LIN {X 0,Y 680.504,Z 396.458,A -85,B 0,C 180,E1 31291.838,E2 31291.838} C_VEL
LIN {X 0,Y 680.503,Z 396.457,A -85,B 0,C 180,E1 31288.855,E2 31288.855} C_VEL
LIN {X 0,Y 680.504,Z 396.449,A -85,B 0,C 180,E1 31285.651,E2 31285.651} C_VEL
LIN {X 0,Y 680.491,Z 396.449,A -85,B 0,C 180,E1 31282.744,E2 31282.744} C_VEL
LIN {X 0,Y 680.522,Z 396.462,A -85,B 0,C 180,E1 31279.612,E2 31279.612} C_VEL
LIN {X 0,Y 680.516,Z 396.57,A -85,B 0,C 180,E1 31279.434,E2 31279.434} C_VEL
LIN {X 0,Y 681.817,Z 400,A -85,B 0,C 180,E1 31279.04,E2 31279.04} C_VEL
LIN {X 0,Y 686.968,Z 410.535,A -85,B 0,C 180,E1 31277.744,E2 31277.744} C_VEL
LIN {X 0,Y 694.908,Z 427.67,A -85,B 0,C 180,E1 31275.744,E2 31275.744} C_VEL
LIN {X 0,Y 695.922,Z 430.045,A -85,B 0,C 180,E1 31275.624,E2 31275.624} C_VEL
LIN {X 0,Y 700.828,Z 449.853,A -85,B 0,C 180,E1 31274.934,E2 31274.934} C_VEL
LIN {X 0,Y 698.454,Z 660.17,A -85,B 0,C 180,E1 31272.2,E2 31272.2} C_VEL
LIN {X 0,Y 696.119,Z 885.552,A -85,B 0,C 180,E1 31269.363,E2 31269.363} C_VEL
LIN {X 0,Y 695.544,Z 917.031,A -85,B 0,C 180,E1 31268.911,E2 31268.911} C_VEL
LIN {X 0,Y 694.786,Z 942.091,A -85,B 0,C 180,E1 31268.4,E2 31268.4} C_VEL
LIN {X 0,Y 693.903,Z 967.65,A -85,B 0,C 180,E1 31267.73,E2 31267.73} C_VEL
LIN {X 0,Y 692.788,Z 994.389,A -85,B 0,C 180,E1 31266.849,E2 31266.849} C_VEL
LIN {X 0,Y 691.794,Z 1015.288,A -85,B 0,C 180,E1 31266.036,E2 31266.036} C_VEL
LIN {X 0,Y 690.754,Z 1035.672,A -85,B 0,C 180,E1 31265.129,E2 31265.129} C_VEL
LIN {X 0,Y 689.674,Z 1055.667,A -85,B 0,C 180,E1 31264.122,E2 31264.122} C_VEL
LIN {X 0,Y 688.501,Z 1076.875,A -85,B 0,C 180,E1 31262.921,E2 31262.921} C_VEL
LIN {X 0,Y 687.033,Z 1101.872,A -85,B 0,C 180,E1 31261.306,E2 31261.306} C_VEL
LIN {X 0,Y 685.952,Z 1121.014,A -85,B 0,C 180,E1 31259.905,E2 31259.905} C_VEL
LIN {X 0,Y 684.924,Z 1139.979,A -85,B 0,C 180,E1 31258.366,E2 31258.366} C_VEL
LIN {X 0,Y 683.775,Z 1160.558,A -85,B 0,C 180,E1 31256.49,E2 31256.49} C_VEL
LIN {X 0,Y 682.966,Z 1177.027,A -85,B 0,C 180,E1 31254.809,E2 31254.809} C_VEL
LIN {X 0,Y 682.152,Z 1194.232,A -85,B 0,C 180,E1 31252.86,E2 31252.86} C_VEL
LIN {X 0,Y 681.475,Z 1210.147,A -85,B 0,C 180,E1 31250.801,E2 31250.801} C_VEL
LIN {X 0,Y 681.039,Z 1222.568,A -85,B 0,C 180,E1 31249.001,E2 31249.001} C_VEL
LIN {X 0,Y 680.648,Z 1234.891,A -85,B 0,C 180,E1 31246.993,E2 31246.993} C_VEL
LIN {X 0,Y 680.343,Z 1246.823,A -85,B 0,C 180,E1 31244.733,E2 31244.733} C_VEL
LIN {X 0,Y 680.159,Z 1255.781,A -85,B 0,C 180,E1 31242.742,E2 31242.742} C_VEL
LIN {X 0,Y 680.022,Z 1262.732,A -85,B 0,C 180,E1 31240.937,E2 31240.937} C_VEL
LIN {X 0,Y 679.93,Z 1268.298,A -85,B 0,C 180,E1 31239.227,E2 31239.227} C_VEL
LIN {X 0,Y 679.925,Z 1273.362,A -85,B 0,C 180,E1 31237.354,E2 31237.354} C_VEL
LIN {X 0,Y 679.917,Z 1277.922,A -85,B 0,C 180,E1 31235.066,E2 31235.066} C_VEL
LIN {X 0,Y 679.912,Z 1280.606,A -85,B 0,C 180,E1 31232.87,E2 31232.87} C_VEL
LIN {X 0,Y 679.875,Z 1281.736,A -85,B 0,C 180,E1 31231.015,E2 31231.015} C_VEL
LIN {X 0,Y 679.863,Z 1281.828,A -85,B 0,C 180,E1 31229.33,E2 31229.33} C_VEL
LIN {X 0,Y 679.906,Z 1280.949,A -85,B 0,C 180,E1 31227.56,E2 31227.56} C_VEL
LIN {X 0,Y 679.915,Z 1278.924,A -85,B 0,C 180,E1 31225.618,E2 31225.618} C_VEL
LIN {X 0,Y 679.927,Z 1274.915,A -85,B 0,C 180,E1 31223.333,E2 31223.333} C_VEL
LIN {X 0,Y 679.942,Z 1269.344,A -85,B 0,C 180,E1 31221.122,E2 31221.122} C_VEL
LIN {X 0,Y 680.018,Z 1263.372,A -85,B 0,C 180,E1 31219.242,E2 31219.242} C_VEL
LIN {X 0,Y 680.138,Z 1256.527,A -85,B 0,C 180,E1 31217.438,E2 31217.438} C_VEL
LIN {X 0,Y 680.303,Z 1248.397,A -85,B 0,C 180,E1 31215.6,E2 31215.6} C_VEL
LIN {X 0,Y 680.526,Z 1238.303,A -85,B 0,C 180,E1 31213.619,E2 31213.619} C_VEL
LIN {X 0,Y 680.965,Z 1224.776,A -85,B 0,C 180,E1 31211.336,E2 31211.336} C_VEL
LIN {X 0,Y 681.406,Z 1211.769,A -85,B 0,C 180,E1 31209.423,E2 31209.423} C_VEL
LIN {X 0,Y 681.966,Z 1198.594,A -85,B 0,C 180,E1 31207.688,E2 31207.688} C_VEL
LIN {X 0,Y 682.779,Z 1180.976,A -85,B 0,C 180,E1 31205.614,E2 31205.614} C_VEL
LIN {X 0,Y 683.632,Z 1163.824,A -85,B 0,C 180,E1 31203.832,E2 31203.832} C_VEL
LIN {X 0,Y 684.496,Z 1146.814,A -85,B 0,C 180,E1 31202.232,E2 31202.232} C_VEL
LIN {X 0,Y 685.785,Z 1124.202,A -85,B 0,C 180,E1 31200.341,E2 31200.341} C_VEL
LIN {X 0,Y 686.861,Z 1105.316,A -85,B 0,C 180,E1 31198.938,E2 31198.938} C_VEL
LIN {X 0,Y 687.97,Z 1085.494,A -85,B 0,C 180,E1 31197.61,E2 31197.61} C_VEL
LIN {X 0,Y 689.434,Z 1060.104,A -85,B 0,C 180,E1 31196.114,E2 31196.114} C_VEL
LIN {X 0,Y 690.588,Z 1038.826,A -85,B 0,C 180,E1 31195.022,E2 31195.022} C_VEL
LIN {X 0,Y 691.614,Z 1018.879,A -85,B 0,C 180,E1 31194.116,E2 31194.116} C_VEL
LIN {X 0,Y 692.522,Z 999.76,A -85,B 0,C 180,E1 31193.35,E2 31193.35} C_VEL
LIN {X 0,Y 693.409,Z 978.617,A -85,B 0,C 180,E1 31192.612,E2 31192.612} C_VEL
LIN {X 0,Y 694.421,Z 953.615,A -85,B 0,C 180,E1 31191.881,E2 31191.881} C_VEL
LIN {X 0,Y 695.3,Z 926.115,A -85,B 0,C 180,E1 31191.258,E2 31191.258} C_VEL
LIN {X 0,Y 695.876,Z 901.264,A -85,B 0,C 180,E1 31190.843,E2 31190.843} C_VEL
LIN {X 0,Y 698.273,Z 676.782,A -85,B 0,C 180,E1 31188.012,E2 31188.012} C_VEL
LIN {X 0,Y 700.623,Z 467.391,A -85,B 0,C 180,E1 31185.297,E2 31185.297} C_VEL
LIN {X 0,Y 700.681,Z 448.554,A -85,B 0,C 180,E1 31185.035,E2 31185.035} C_VEL
LIN {X 0,Y 695.292,Z 428.27,A -85,B 0,C 180,E1 31184.297,E2 31184.297} C_VEL
LIN {X 0,Y 693.526,Z 424.504,A -85,B 0,C 180,E1 31183.907,E2 31183.907} C_VEL
LIN {X 0,Y 684.276,Z 404.782,A -85,B 0,C 180,E1 31181.56,E2 31181.56} C_VEL
LIN {X 0,Y 681.818,Z 399.996,A -85,B 0,C 180,E1 31180.96,E2 31180.96} C_VEL
LIN {X 0,Y 680.501,Z 396.443,A -85,B 0,C 180,E1 31180.523,E2 31180.523} C_VEL
LIN {X 0,Y 680.481,Z 396.449,A -85,B 0,C 180,E1 31177.469,E2 31177.469} C_VEL
LIN {X 0,Y 680.464,Z 396.461,A -85,B 0,C 180,E1 31174.76,E2 31174.76} C_VEL
LIN {X 0,Y 680.524,Z 396.466,A -85,B 0,C 180,E1 31171.723,E2 31171.723} C_VEL
LIN {X 0,Y 680.451,Z 396.462,A -85,B 0,C 180,E1 31168.911,E2 31168.911} C_VEL
LIN {X 0,Y 680.472,Z 396.462,A -85,B 0,C 180,E1 31166.25,E2 31166.25} C_VEL
LIN {X 0,Y 680.462,Z 396.469,A -85,B 0,C 180,E1 31163.1,E2 31163.1} C_VEL
LIN {X 0,Y 680.435,Z 396.45,A -85,B 0,C 180,E1 31160.561,E2 31160.561} C_VEL
LIN {X 0,Y 680.475,Z 396.464,A -85,B 0,C 180,E1 31157.885,E2 31157.885} C_VEL
LIN {X 0,Y 680.439,Z 396.45,A -85,B 0,C 180,E1 31154.807,E2 31154.807} C_VEL
LIN {X 0,Y 680.422,Z 396.468,A -85,B 0,C 180,E1 31152.389,E2 31152.389} C_VEL
LIN {X 0,Y 680.443,Z 396.458,A -85,B 0,C 180,E1 31149.815,E2 31149.815} C_VEL
LIN {X 0,Y 680.436,Z 396.47,A -85,B 0,C 180,E1 31146.663,E2 31146.663} C_VEL
LIN {X 0,Y 680.418,Z 396.459,A -85,B 0,C 180,E1 31144.129,E2 31144.129} C_VEL
LIN {X 0,Y 680.469,Z 396.458,A -85,B 0,C 180,E1 31141.431,E2 31141.431} C_VEL
LIN {X 0,Y 680.444,Z 396.457,A -85,B 0,C 180,E1 31138.4,E2 31138.4} C_VEL
LIN {X 0,Y 680.433,Z 396.456,A -85,B 0,C 180,E1 31135.871,E2 31135.871} C_VEL
LIN {X 0,Y 680.507,Z 396.463,A -85,B 0,C 180,E1 31133.08,E2 31133.08} C_VEL
LIN {X 0,Y 680.451,Z 396.455,A -85,B 0,C 180,E1 31130.1,E2 31130.1} C_VEL
LIN {X 0,Y 680.452,Z 396.467,A -85,B 0,C 180,E1 31127.525,E2 31127.525} C_VEL
LIN {X 0,Y 680.527,Z 396.444,A -85,B 0,C 180,E1 31124.577,E2 31124.577} C_VEL
LIN {X 0,Y 680.457,Z 396.464,A -85,B 0,C 180,E1 31121.672,E2 31121.672} C_VEL
LIN {X 0,Y 680.499,Z 396.445,A -85,B 0,C 180,E1 31118.894,E2 31118.894} C_VEL
LIN {X 0,Y 680.478,Z 396.458,A -85,B 0,C 180,E1 31115.797,E2 31115.797} C_VEL
LIN {X 0,Y 680.475,Z 396.456,A -85,B 0,C 180,E1 31113.091,E2 31113.091} C_VEL
LIN {X 0,Y 680.53,Z 396.439,A -85,B 0,C 180,E1 31110.029,E2 31110.029} C_VEL
LIN {X 0,Y 680.473,Z 396.445,A -85,B 0,C 180,E1 31109.296,E2 31109.296} C_VEL
LIN {X 0,Y 679.489,Z 396.577,A -85,B 0,C 180,E1 31108.648,E2 31108.648} C_VEL
LIN {X 0,Y 673.118,Z 397.384,A -85,B 0,C 180,E1 31106.83,E2 31106.83} C_VEL
LIN {X 0,Y 672.585,Z 397.437,A -85,B 0,C 180,E1 31106.358,E2 31106.358} C_VEL
LIN {X 0,Y 672.547,Z 397.454,A -85,B 0,C 180,E1 31103.297,E2 31103.297} C_VEL
LIN {X 0,Y 672.585,Z 397.443,A -85,B 0,C 180,E1 31100.351,E2 31100.351} C_VEL
LIN {X 0,Y 672.605,Z 397.605,A -85,B 0,C 180,E1 31097.725,E2 31097.725} C_VEL
LIN {X 0,Y 674.077,Z 401.205,A -85,B 0,C 180,E1 31097.494,E2 31097.494} C_VEL
LIN {X 0,Y 676.461,Z 403.778,A -85,B 0,C 180,E1 31097.233,E2 31097.233} C_VEL
LIN {X 0,Y 679.086,Z 407.676,A -85,B 0,C 180,E1 31096.935,E2 31096.935} C_VEL
LIN {X 0,Y 689.098,Z 422.003,A -85,B 0,C 180,E1 31095.839,E2 31095.839} C_VEL
LIN {X 0,Y 694.997,Z 431.183,A -85,B 0,C 180,E1 31095.208,E2 31095.208} C_VEL
LIN {X 0,Y 692.464,Z 634.839,A -85,B 0,C 180,E1 31092.542,E2 31092.542} C_VEL
LIN {X 0,Y 689.877,Z 860.243,A -85,B 0,C 180,E1 31089.682,E2 31089.682} C_VEL
LIN {X 0,Y 689.241,Z 888.714,A -85,B 0,C 180,E1 31089.255,E2 31089.255} C_VEL
LIN {X 0,Y 688.441,Z 912.912,A -85,B 0,C 180,E1 31088.753,E2 31088.753} C_VEL
LIN {X 0,Y 687.432,Z 939.222,A -85,B 0,C 180,E1 31088.053,E2 31088.053} C_VEL
LIN {X 0,Y 686.198,Z 965.515,A -85,B 0,C 180,E1 31087.172,E2 31087.172} C_VEL
LIN {X 0,Y 685.083,Z 986.774,A -85,B 0,C 180,E1 31086.332,E2 31086.332} C_VEL
LIN {X 0,Y 683.941,Z 1006.966,A -85,B 0,C 180,E1 31085.42,E2 31085.42} C_VEL
LIN {X 0,Y 682.713,Z 1027.539,A -85,B 0,C 180,E1 31084.367,E2 31084.367} C_VEL
LIN {X 0,Y 681.185,Z 1052.091,A -85,B 0,C 180,E1 31082.939,E2 31082.939} C_VEL
LIN {X 0,Y 679.791,Z 1073.383,A -85,B 0,C 180,E1 31081.52,E2 31081.52} C_VEL
LIN {X 0,Y 678.624,Z 1092.09,A -85,B 0,C 180,E1 31080.129,E2 31080.129} C_VEL
LIN {X 0,Y 677.353,Z 1113.291,A -85,B 0,C 180,E1 31078.374,E2 31078.374} C_VEL
LIN {X 0,Y 676.173,Z 1132.066,A -85,B 0,C 180,E1 31076.613,E2 31076.613} C_VEL
LIN {X 0,Y 675.296,Z 1148.032,A -85,B 0,C 180,E1 31074.954,E2 31074.954} C_VEL
LIN {X 0,Y 674.34,Z 1166.118,A -85,B 0,C 180,E1 31072.855,E2 31072.855} C_VEL
LIN {X 0,Y 673.669,Z 1180.534,A -85,B 0,C 180,E1 31070.954,E2 31070.954} C_VEL
LIN {X 0,Y 673.181,Z 1192.813,A -85,B 0,C 180,E1 31069.149,E2 31069.149} C_VEL
LIN {X 0,Y 672.723,Z 1205.66,A -85,B 0,C 180,E1 31067.021,E2 31067.021} C_VEL
LIN {X 0,Y 672.382,Z 1217.474,A -85,B 0,C 180,E1 31064.727,E2 31064.727} C_VEL
LIN {X 0,Y 672.187,Z 1225.987,A -85,B 0,C 180,E1 31062.801,E2 31062.801} C_VEL
LIN {X 0,Y 672.041,Z 1232.908,A -85,B 0,C 180,E1 31060.974,E2 31060.974} C_VEL
LIN {X 0,Y 671.938,Z 1238.444,A -85,B 0,C 180,E1 31059.244,E2 31059.244} C_VEL
LIN {X 0,Y 671.926,Z 1243.472,A -85,B 0,C 180,E1 31057.348,E2 31057.348} C_VEL
LIN {X 0,Y 671.919,Z 1247.993,A -85,B 0,C 180,E1 31055.033,E2 31055.033} C_VEL
LIN {X 0,Y 671.912,Z 1250.644,A -85,B 0,C 180,E1 31052.811,E2 31052.811} C_VEL
LIN {X 0,Y 671.874,Z 1251.749,A -85,B 0,C 180,E1 31050.934,E2 31050.934} C_VEL
LIN {X 0,Y 671.863,Z 1251.815,A -85,B 0,C 180,E1 31049.229,E2 31049.229} C_VEL
LIN {X 0,Y 671.904,Z 1250.912,A -85,B 0,C 180,E1 31047.437,E2 31047.437} C_VEL
LIN {X 0,Y 671.912,Z 1248.858,A -85,B 0,C 180,E1 31045.473,E2 31045.473} C_VEL
LIN {X 0,Y 671.928,Z 1244.818,A -85,B 0,C 180,E1 31043.159,E2 31043.159} C_VEL
LIN {X 0,Y 671.944,Z 1239.453,A -85,B 0,C 180,E1 31041.008,E2 31041.008} C_VEL
LIN {X 0,Y 672.028,Z 1233.504,A -85,B 0,C 180,E1 31039.105,E2 31039.105} C_VEL
LIN {X 0,Y 672.179,Z 1226.323,A -85,B 0,C 180,E1 31037.191,E2 31037.191} C_VEL
LIN {X 0,Y 672.363,Z 1218.266,A -85,B 0,C 180,E1 31035.353,E2 31035.353} C_VEL
LIN {X 0,Y 672.625,Z 1208.03,A -85,B 0,C 180,E1 31033.324,E2 31033.324} C_VEL
LIN {X 0,Y 673.12,Z 1194.433,A -85,B 0,C 180,E1 31031.012,E2 31031.012} C_VEL
LIN {X 0,Y 673.609,Z 1181.757,A -85,B 0,C 180,E1 31029.127,E2 31029.127} C_VEL
LIN {X 0,Y 674.248,Z 1167.886,A -85,B 0,C 180,E1 31027.281,E2 31027.281} C_VEL
LIN {X 0,Y 675.222,Z 1149.613,A -85,B 0,C 180,E1 31025.128,E2 31025.128} C_VEL
LIN {X 0,Y 676.126,Z 1132.865,A -85,B 0,C 180,E1 31023.376,E2 31023.376} C_VEL
LIN {X 0,Y 677.209,Z 1115.165,A -85,B 0,C 180,E1 31021.706,E2 31021.706} C_VEL
LIN {X 0,Y 678.547,Z 1093.392,A -85,B 0,C 180,E1 31019.882,E2 31019.882} C_VEL
LIN {X 0,Y 679.733,Z 1074.478,A -85,B 0,C 180,E1 31018.468,E2 31018.468} C_VEL
LIN {X 0,Y 681.034,Z 1054.017,A -85,B 0,C 180,E1 31017.094,E2 31017.094} C_VEL
LIN {X 0,Y 682.632,Z 1028.954,A -85,B 0,C 180,E1 31015.619,E2 31015.619} C_VEL
LIN {X 0,Y 683.91,Z 1007.528,A -85,B 0,C 180,E1 31014.518,E2 31014.518} C_VEL
LIN {X 0,Y 685.049,Z 987.394,A -85,B 0,C 180,E1 31013.605,E2 31013.605} C_VEL
LIN {X 0,Y 686.095,Z 967.48,A -85,B 0,C 180,E1 31012.812,E2 31012.812} C_VEL
LIN {X 0,Y 687.136,Z 945.081,A -85,B 0,C 180,E1 31012.04,E2 31012.04} C_VEL
LIN {X 0,Y 688.28,Z 918.034,A -85,B 0,C 180,E1 31011.278,E2 31011.278} C_VEL
LIN {X 0,Y 689.111,Z 892.431,A -85,B 0,C 180,E1 31010.723,E2 31010.723} C_VEL
LIN {X 0,Y 689.749,Z 867.404,A -85,B 0,C 180,E1 31010.322,E2 31010.322} C_VEL
LIN {X 0,Y 692.38,Z 641.833,A -85,B 0,C 180,E1 31007.458,E2 31007.458} C_VEL
LIN {X 0,Y 694.953,Z 435.033,A -85,B 0,C 180,E1 31004.754,E2 31004.754} C_VEL
LIN {X 0,Y 694.842,Z 430.636,A -85,B 0,C 180,E1 31004.681,E2 31004.681} C_VEL
LIN {X 0,Y 682.15,Z 411.898,A -85,B 0,C 180,E1 31003.314,E2 31003.314} C_VEL
LIN {X 0,Y 678.641,Z 407.17,A -85,B 0,C 180,E1 31002.927,E2 31002.927} C_VEL
LIN {X 0,Y 675.796,Z 402.92,A -85,B 0,C 180,E1 31002.603,E2 31002.603} C_VEL
LIN {X 0,Y 673.436,Z 400.174,A -85,B 0,C 180,E1 31002.34,E2 31002.34} C_VEL
LIN {X 0,Y 672.594,Z 397.588,A -85,B 0,C 180,E1 31002.182,E2 31002.182} C_VEL
LIN {X 0,Y 672.576,Z 397.451,A -85,B 0,C 180,E1 30999.099,E2 30999.099} C_VEL
LIN {X 0,Y 672.576,Z 397.449,A -85,B 0,C 180,E1 30996.025,E2 30996.025} C_VEL
LIN {X 0,Y 672.581,Z 397.45,A -85,B 0,C 180,E1 30992.964,E2 30992.964} C_VEL
LIN {X 0,Y 672.58,Z 397.429,A -85,B 0,C 180,E1 30989.87,E2 30989.87} C_VEL
LIN {X 0,Y 672.582,Z 397.439,A -85,B 0,C 180,E1 30986.773,E2 30986.773} C_VEL
LIN {X 0,Y 672.579,Z 397.444,A -85,B 0,C 180,E1 30983.666,E2 30983.666} C_VEL
LIN {X 0,Y 672.58,Z 397.43,A -85,B 0,C 180,E1 30980.539,E2 30980.539} C_VEL
LIN {X 0,Y 672.573,Z 397.447,A -85,B 0,C 180,E1 30977.387,E2 30977.387} C_VEL
LIN {X 0,Y 672.584,Z 397.43,A -85,B 0,C 180,E1 30974.287,E2 30974.287} C_VEL
LIN {X 0,Y 672.569,Z 397.446,A -85,B 0,C 180,E1 30971.144,E2 30971.144} C_VEL
LIN {X 0,Y 672.582,Z 397.432,A -85,B 0,C 180,E1 30968.033,E2 30968.033} C_VEL
LIN {X 0,Y 672.57,Z 397.445,A -85,B 0,C 180,E1 30964.947,E2 30964.947} C_VEL
LIN {X 0,Y 672.579,Z 397.431,A -85,B 0,C 180,E1 30961.874,E2 30961.874} C_VEL
LIN {X 0,Y 672.574,Z 397.444,A -85,B 0,C 180,E1 30958.807,E2 30958.807} C_VEL
LIN {X 0,Y 672.575,Z 397.43,A -85,B 0,C 180,E1 30955.737,E2 30955.737} C_VEL
LIN {X 0,Y 672.57,Z 397.442,A -85,B 0,C 180,E1 30952.569,E2 30952.569} C_VEL
LIN {X 0,Y 672.579,Z 397.436,A -85,B 0,C 180,E1 30949.464,E2 30949.464} C_VEL
LIN {X 0,Y 672.566,Z 397.439,A -85,B 0,C 180,E1 30946.327,E2 30946.327} C_VEL
LIN {X 0,Y 672.573,Z 397.445,A -85,B 0,C 180,E1 30943.326,E2 30943.326} C_VEL
LIN {X 0,Y 672.571,Z 397.429,A -85,B 0,C 180,E1 30940.186,E2 30940.186} C_VEL
LIN {X 0,Y 672.566,Z 397.455,A -85,B 0,C 180,E1 30937.168,E2 30937.168} C_VEL
LIN {X 0,Y 672.571,Z 397.44,A -85,B 0,C 180,E1 30933.987,E2 30933.987} C_VEL
LIN {X 0,Y 672.555,Z 397.442,A -85,B 0,C 180,E1 30931.009,E2 30931.009} C_VEL
LIN {X 0,Y 672.576,Z 397.448,A -85,B 0,C 180,E1 30927.844,E2 30927.844} C_VEL
LIN {X 0,Y 672.552,Z 397.448,A -85,B 0,C 180,E1 30924.856,E2 30924.856} C_VEL
LIN {X 0,Y 672.582,Z 397.438,A -85,B 0,C 180,E1 30921.718,E2 30921.718} C_VEL
LIN {X 0,Y 672.591,Z 397.507,A -85,B 0,C 180,E1 30920.121,E2 30920.121} C_VEL
LIN {X 0,Y 673.604,Z 400.471,A -85,B 0,C 180,E1 30919.781,E2 30919.781} C_VEL
LIN {X 0,Y 674.827,Z 402.796,A -85,B 0,C 180,E1 30919.476,E2 30919.476} C_VEL
LIN {X 0,Y 682.843,Z 419.415,A -85,B 0,C 180,E1 30917.428,E2 30917.428} C_VEL
LIN {X 0,Y 686.977,Z 428.148,A -85,B 0,C 180,E1 30916.42,E2 30916.42} C_VEL
LIN {X 0,Y 690.759,Z 434.1,A -85,B 0,C 180,E1 30916.004,E2 30916.004} C_VEL
LIN {X 0,Y 695.129,Z 451.991,A -85,B 0,C 180,E1 30915.374,E2 30915.374} C_VEL
LIN {X 0,Y 692.503,Z 661.697,A -85,B 0,C 180,E1 30912.627,E2 30912.627} C_VEL
LIN {X 0,Y 689.911,Z 887.155,A -85,B 0,C 180,E1 30909.765,E2 30909.765} C_VEL
LIN {X 0,Y 689.28,Z 917.493,A -85,B 0,C 180,E1 30909.322,E2 30909.322} C_VEL
LIN {X 0,Y 688.472,Z 942.07,A -85,B 0,C 180,E1 30908.818,E2 30908.818} C_VEL
LIN {X 0,Y 687.49,Z 967.641,A -85,B 0,C 180,E1 30908.145,E2 30908.145} C_VEL
LIN {X 0,Y 686.228,Z 994.964,A -85,B 0,C 180,E1 30907.237,E2 30907.237} C_VEL
LIN {X 0,Y 685.1,Z 1016.414,A -85,B 0,C 180,E1 30906.392,E2 30906.392} C_VEL
LIN {X 0,Y 683.959,Z 1036.657,A -85,B 0,C 180,E1 30905.48,E2 30905.48} C_VEL
LIN {X 0,Y 682.729,Z 1057.275,A -85,B 0,C 180,E1 30904.427,E2 30904.427} C_VEL
LIN {X 0,Y 681.203,Z 1081.887,A -85,B 0,C 180,E1 30902.997,E2 30902.997} C_VEL
LIN {X 0,Y 679.766,Z 1103.872,A -85,B 0,C 180,E1 30901.531,E2 30901.531} C_VEL
LIN {X 0,Y 678.586,Z 1122.741,A -85,B 0,C 180,E1 30900.124,E2 30900.124} C_VEL
LIN {X 0,Y 677.319,Z 1143.765,A -85,B 0,C 180,E1 30898.376,E2 30898.376} C_VEL
LIN {X 0,Y 676.152,Z 1162.422,A -85,B 0,C 180,E1 30896.623,E2 30896.623} C_VEL
LIN {X 0,Y 675.281,Z 1178.361,A -85,B 0,C 180,E1 30894.964,E2 30894.964} C_VEL
LIN {X 0,Y 674.324,Z 1196.4,A -85,B 0,C 180,E1 30892.864,E2 30892.864} C_VEL
LIN {X 0,Y 673.655,Z 1210.793,A -85,B 0,C 180,E1 30890.963,E2 30890.963} C_VEL
LIN {X 0,Y 673.152,Z 1223.573,A -85,B 0,C 180,E1 30889.077,E2 30889.077} C_VEL
LIN {X 0,Y 672.652,Z 1237.329,A -85,B 0,C 180,E1 30886.764,E2 30886.764} C_VEL
LIN {X 0,Y 672.367,Z 1248.056,A -85,B 0,C 180,E1 30884.647,E2 30884.647} C_VEL
LIN {X 0,Y 672.177,Z 1256.497,A -85,B 0,C 180,E1 30882.721,E2 30882.721} C_VEL
LIN {X 0,Y 672.03,Z 1263.651,A -85,B 0,C 180,E1 30880.809,E2 30880.809} C_VEL
LIN {X 0,Y 671.974,Z 1270.806,A -85,B 0,C 180,E1 30878.475,E2 30878.475} C_VEL
LIN {X 0,Y 671.931,Z 1276.089,A -85,B 0,C 180,E1 30876.154,E2 30876.154} C_VEL
LIN {X 0,Y 671.915,Z 1279.581,A -85,B 0,C 180,E1 30873.929,E2 30873.929} C_VEL
LIN {X 0,Y 671.908,Z 1281.623,A -85,B 0,C 180,E1 30871.453,E2 30871.453} C_VEL
LIN {X 0,Y 671.865,Z 1281.85,A -85,B 0,C 180,E1 30869.407,E2 30869.407} C_VEL
LIN {X 0,Y 671.907,Z 1281.017,A -85,B 0,C 180,E1 30867.616,E2 30867.616} C_VEL
LIN {X 0,Y 671.914,Z 1278.96,A -85,B 0,C 180,E1 30865.595,E2 30865.595} C_VEL
LIN {X 0,Y 671.93,Z 1274.915,A -85,B 0,C 180,E1 30863.253,E2 30863.253} C_VEL
LIN {X 0,Y 671.942,Z 1269.344,A -85,B 0,C 180,E1 30861.015,E2 30861.015} C_VEL
LIN {X 0,Y 672.033,Z 1263.362,A -85,B 0,C 180,E1 30859.11,E2 30859.11} C_VEL
LIN {X 0,Y 672.183,Z 1256.171,A -85,B 0,C 180,E1 30857.199,E2 30857.199} C_VEL
LIN {X 0,Y 672.378,Z 1247.683,A -85,B 0,C 180,E1 30855.273,E2 30855.273} C_VEL
LIN {X 0,Y 672.716,Z 1235.92,A -85,B 0,C 180,E1 30852.979,E2 30852.979} C_VEL
LIN {X 0,Y 673.174,Z 1223.046,A -85,B 0,C 180,E1 30850.842,E2 30850.842} C_VEL
LIN {X 0,Y 673.667,Z 1210.545,A -85,B 0,C 180,E1 30849.003,E2 30849.003} C_VEL
LIN {X 0,Y 674.405,Z 1195.043,A -85,B 0,C 180,E1 30846.963,E2 30846.963} C_VEL
LIN {X 0,Y 675.313,Z 1177.593,A -85,B 0,C 180,E1 30844.953,E2 30844.953} C_VEL
LIN {X 0,Y 676.197,Z 1161.576,A -85,B 0,C 180,E1 30843.293,E2 30843.293} C_VEL
LIN {X 0,Y 677.462,Z 1141.497,A -85,B 0,C 180,E1 30841.424,E2 30841.424} C_VEL
LIN {X 0,Y 678.645,Z 1121.729,A -85,B 0,C 180,E1 30839.798,E2 30839.798} C_VEL
LIN {X 0,Y 679.798,Z 1103.323,A -85,B 0,C 180,E1 30838.431,E2 30838.431} C_VEL
LIN {X 0,Y 681.311,Z 1080.545,A -85,B 0,C 180,E1 30836.917,E2 30836.917} C_VEL
LIN {X 0,Y 682.766,Z 1056.612,A -85,B 0,C 180,E1 30835.538,E2 30835.538} C_VEL
LIN {X 0,Y 683.963,Z 1036.584,A -85,B 0,C 180,E1 30834.517,E2 30834.517} C_VEL
LIN {X 0,Y 685.09,Z 1016.623,A -85,B 0,C 180,E1 30833.617,E2 30833.617} C_VEL
LIN {X 0,Y 686.179,Z 995.905,A -85,B 0,C 180,E1 30832.798,E2 30832.798} C_VEL
LIN {X 0,Y 687.419,Z 969.551,A -85,B 0,C 180,E1 30831.912,E2 30831.912} C_VEL
LIN {X 0,Y 688.433,Z 943.106,A -85,B 0,C 180,E1 30831.206,E2 30831.206} C_VEL
LIN {X 0,Y 689.236,Z 918.781,A -85,B 0,C 180,E1 30830.701,E2 30830.701} C_VEL
LIN {X 0,Y 689.874,Z 890.444,A -85,B 0,C 180,E1 30830.276,E2 30830.276} C_VEL
LIN {X 0,Y 692.469,Z 664.525,A -85,B 0,C 180,E1 30827.409,E2 30827.409} C_VEL
LIN {X 0,Y 695.106,Z 453.752,A -85,B 0,C 180,E1 30824.649,E2 30824.649} C_VEL
LIN {X 0,Y 694.92,Z 450.484,A -85,B 0,C 180,E1 30824.587,E2 30824.587} C_VEL
LIN {X 0,Y 690.338,Z 433.14,A -85,B 0,C 180,E1 30823.945,E2 30823.945} C_VEL
LIN {X 0,Y 686.543,Z 427.36,A -85,B 0,C 180,E1 30823.516,E2 30823.516} C_VEL
LIN {X 0,Y 678.406,Z 410.05,A -85,B 0,C 180,E1 30821.435,E2 30821.435} C_VEL
LIN {X 0,Y 674.576,Z 401.892,A -85,B 0,C 180,E1 30820.428,E2 30820.428} C_VEL
LIN {X 0,Y 672.72,Z 398.195,A -85,B 0,C 180,E1 30819.949,E2 30819.949} C_VEL
LIN {X 0,Y 672.584,Z 397.438,A -85,B 0,C 180,E1 30819.847,E2 30819.847} C_VEL
LIN {X 0,Y 672.521,Z 397.442,A -85,B 0,C 180,E1 30817.024,E2 30817.024} C_VEL
LIN {X 0,Y 672.576,Z 397.434,A -85,B 0,C 180,E1 30814.191,E2 30814.191} C_VEL
LIN {X 0,Y 672.523,Z 397.451,A -85,B 0,C 180,E1 30811.158,E2 30811.158} C_VEL
LIN {X 0,Y 672.517,Z 397.449,A -85,B 0,C 180,E1 30808.53,E2 30808.53} C_VEL
LIN {X 0,Y 672.573,Z 397.433,A -85,B 0,C 180,E1 30805.54,E2 30805.54} C_VEL
LIN {X 0,Y 672.502,Z 397.457,A -85,B 0,C 180,E1 30802.742,E2 30802.742} C_VEL
LIN {X 0,Y 672.512,Z 397.435,A -85,B 0,C 180,E1 30800.178,E2 30800.178} C_VEL
LIN {X 0,Y 672.522,Z 397.454,A -85,B 0,C 180,E1 30797.031,E2 30797.031} C_VEL
LIN {X 0,Y 672.486,Z 397.44,A -85,B 0,C 180,E1 30794.465,E2 30794.465} C_VEL
LIN {X 0,Y 672.505,Z 397.457,A -85,B 0,C 180,E1 30791.927,E2 30791.927} C_VEL
LIN {X 0,Y 672.496,Z 397.441,A -85,B 0,C 180,E1 30788.723,E2 30788.723} C_VEL
LIN {X 0,Y 672.477,Z 397.459,A -85,B 0,C 180,E1 30786.231,E2 30786.231} C_VEL
LIN {X 0,Y 672.504,Z 397.442,A -85,B 0,C 180,E1 30783.666,E2 30783.666} C_VEL
LIN {X 0,Y 672.508,Z 397.457,A -85,B 0,C 180,E1 30780.511,E2 30780.511} C_VEL
LIN {X 0,Y 672.49,Z 397.446,A -85,B 0,C 180,E1 30777.955,E2 30777.955} C_VEL
LIN {X 0,Y 672.561,Z 397.446,A -85,B 0,C 180,E1 30775.139,E2 30775.139} C_VEL
LIN {X 0,Y 672.508,Z 397.443,A -85,B 0,C 180,E1 30772.138,E2 30772.138} C_VEL
LIN {X 0,Y 672.51,Z 397.445,A -85,B 0,C 180,E1 30769.549,E2 30769.549} C_VEL
LIN {X 0,Y 672.589,Z 397.438,A -85,B 0,C 180,E1 30766.59,E2 30766.59} C_VEL
LIN {X 0,Y 672.516,Z 397.446,A -85,B 0,C 180,E1 30763.769,E2 30763.769} C_VEL
LIN {X 0,Y 672.543,Z 397.453,A -85,B 0,C 180,E1 30761.088,E2 30761.088} C_VEL
LIN {X 0,Y 672.542,Z 397.449,A -85,B 0,C 180,E1 30757.905,E2 30757.905} C_VEL
LIN {X 0,Y 672.53,Z 397.447,A -85,B 0,C 180,E1 30755.212,E2 30755.212} C_VEL
LIN {X 0,Y 672.591,Z 397.45,A -85,B 0,C 180,E1 30752.173,E2 30752.173} C_VEL
LIN {X 0,Y 672.533,Z 397.433,A -85,B 0,C 180,E1 30749.23,E2 30749.23} C_VEL
LIN {X 0,Y 672.585,Z 397.437,A -85,B 0,C 180,E1 30746.358,E2 30746.358} C_VEL
LIN {X 0,Y 671.592,Z 397.553,A -85,B 0,C 180,E1 30745.701,E2 30745.701} C_VEL
LIN {X 0,Y 665.164,Z 398.376,A -85,B 0,C 180,E1 30743.862,E2 30743.862} C_VEL
LIN {X 0,Y 664.613,Z 398.443,A -85,B 0,C 180,E1 30743.384,E2 30743.384} C_VEL
LIN {X 0,Y 664.647,Z 398.431,A -85,B 0,C 180,E1 30740.366,E2 30740.366} C_VEL
LIN {X 0,Y 664.66,Z 398.582,A -85,B 0,C 180,E1 30738.438,E2 30738.438} C_VEL
LIN {X 0,Y 665.854,Z 401.773,A -85,B 0,C 180,E1 30738.27,E2 30738.27} C_VEL
LIN {X 0,Y 668.717,Z 404.963,A -85,B 0,C 180,E1 30737.943,E2 30737.943} C_VEL
LIN {X 0,Y 671.372,Z 408.83,A -85,B 0,C 180,E1 30737.629,E2 30737.629} C_VEL
LIN {X 0,Y 673.017,Z 411.059,A -85,B 0,C 180,E1 30737.44,E2 30737.44} C_VEL
LIN {X 0,Y 681.12,Z 422.27,A -85,B 0,C 180,E1 30736.532,E2 30736.532} C_VEL
LIN {X 0,Y 689.306,Z 434.97,A -85,B 0,C 180,E1 30735.632,E2 30735.632} C_VEL
LIN {X 0,Y 686.515,Z 638.897,A -85,B 0,C 180,E1 30732.943,E2 30732.943} C_VEL
LIN {X 0,Y 683.643,Z 864.967,A -85,B 0,C 180,E1 30730.05,E2 30730.05} C_VEL
LIN {X 0,Y 682.944,Z 890.972,A -85,B 0,C 180,E1 30729.641,E2 30729.641} C_VEL
LIN {X 0,Y 682.071,Z 915.262,A -85,B 0,C 180,E1 30729.123,E2 30729.123} C_VEL
LIN {X 0,Y 680.927,Z 941.935,A -85,B 0,C 180,E1 30728.392,E2 30728.392} C_VEL
LIN {X 0,Y 679.661,Z 966.228,A -85,B 0,C 180,E1 30727.562,E2 30727.562} C_VEL
LIN {X 0,Y 678.477,Z 986.785,A -85,B 0,C 180,E1 30726.743,E2 30726.743} C_VEL
LIN {X 0,Y 677.229,Z 1006.977,A -85,B 0,C 180,E1 30725.825,E2 30725.825} C_VEL
LIN {X 0,Y 675.831,Z 1028.443,A -85,B 0,C 180,E1 30724.716,E2 30724.716} C_VEL
LIN {X 0,Y 674.078,Z 1053.761,A -85,B 0,C 180,E1 30723.216,E2 30723.216} C_VEL
LIN {X 0,Y 672.624,Z 1074.057,A -85,B 0,C 180,E1 30721.845,E2 30721.845} C_VEL
LIN {X 0,Y 671.318,Z 1093.053,A -85,B 0,C 180,E1 30720.414,E2 30720.414} C_VEL
LIN {X 0,Y 669.857,Z 1114.821,A -85,B 0,C 180,E1 30718.575,E2 30718.575} C_VEL
LIN {X 0,Y 668.644,Z 1132.538,A -85,B 0,C 180,E1 30716.889,E2 30716.889} C_VEL
LIN {X 0,Y 667.667,Z 1148.232,A -85,B 0,C 180,E1 30715.237,E2 30715.237} C_VEL
LIN {X 0,Y 666.638,Z 1166.125,A -85,B 0,C 180,E1 30713.134,E2 30713.134} C_VEL
LIN {X 0,Y 665.874,Z 1180.823,A -85,B 0,C 180,E1 30711.17,E2 30711.17} C_VEL
LIN {X 0,Y 665.316,Z 1193.369,A -85,B 0,C 180,E1 30709.298,E2 30709.298} C_VEL
LIN {X 0,Y 664.789,Z 1206.677,A -85,B 0,C 180,E1 30707.05,E2 30707.05} C_VEL
LIN {X 0,Y 664.428,Z 1217.888,A -85,B 0,C 180,E1 30704.818,E2 30704.818} C_VEL
LIN {X 0,Y 664.212,Z 1226.348,A -85,B 0,C 180,E1 30702.868,E2 30702.868} C_VEL
LIN {X 0,Y 664.051,Z 1233.522,A -85,B 0,C 180,E1 30700.932,E2 30700.932} C_VEL
LIN {X 0,Y 663.97,Z 1240.483,A -85,B 0,C 180,E1 30698.657,E2 30698.657} C_VEL
LIN {X 0,Y 663.934,Z 1246.018,A -85,B 0,C 180,E1 30696.221,E2 30696.221} C_VEL
LIN {X 0,Y 663.915,Z 1249.537,A -85,B 0,C 180,E1 30693.968,E2 30693.968} C_VEL
LIN {X 0,Y 663.909,Z 1251.613,A -85,B 0,C 180,E1 30691.463,E2 30691.463} C_VEL
LIN {X 0,Y 663.866,Z 1251.86,A -85,B 0,C 180,E1 30689.392,E2 30689.392} C_VEL
LIN {X 0,Y 663.903,Z 1251.046,A -85,B 0,C 180,E1 30687.579,E2 30687.579} C_VEL
LIN {X 0,Y 663.915,Z 1249.053,A -85,B 0,C 180,E1 30685.569,E2 30685.569} C_VEL
LIN {X 0,Y 663.93,Z 1245.16,A -85,B 0,C 180,E1 30683.25,E2 30683.25} C_VEL
LIN {X 0,Y 663.949,Z 1239.705,A -85,B 0,C 180,E1 30680.986,E2 30680.986} C_VEL
LIN {X 0,Y 664.046,Z 1233.503,A -85,B 0,C 180,E1 30678.972,E2 30678.972} C_VEL
LIN {X 0,Y 664.211,Z 1226.322,A -85,B 0,C 180,E1 30677.035,E2 30677.035} C_VEL
LIN {X 0,Y 664.416,Z 1218.264,A -85,B 0,C 180,E1 30675.174,E2 30675.174} C_VEL
LIN {X 0,Y 664.735,Z 1207.779,A -85,B 0,C 180,E1 30673.072,E2 30673.072} C_VEL
LIN {X 0,Y 665.296,Z 1193.854,A -85,B 0,C 180,E1 30670.689,E2 30670.689} C_VEL
LIN {X 0,Y 665.86,Z 1181.11,A -85,B 0,C 180,E1 30668.78,E2 30668.78} C_VEL
LIN {X 0,Y 666.644,Z 1166.033,A -85,B 0,C 180,E1 30666.764,E2 30666.764} C_VEL
LIN {X 0,Y 667.642,Z 1148.76,A -85,B 0,C 180,E1 30664.731,E2 30664.731} C_VEL
LIN {X 0,Y 668.628,Z 1132.681,A -85,B 0,C 180,E1 30663.035,E2 30663.035} C_VEL
LIN {X 0,Y 669.912,Z 1114.142,A -85,B 0,C 180,E1 30661.272,E2 30661.272} C_VEL
LIN {X 0,Y 671.337,Z 1092.775,A -85,B 0,C 180,E1 30659.474,E2 30659.474} C_VEL
LIN {X 0,Y 672.643,Z 1073.801,A -85,B 0,C 180,E1 30658.046,E2 30658.046} C_VEL
LIN {X 0,Y 674.247,Z 1051.799,A -85,B 0,C 180,E1 30656.567,E2 30656.567} C_VEL
LIN {X 0,Y 675.91,Z 1027.164,A -85,B 0,C 180,E1 30655.125,E2 30655.125} C_VEL
LIN {X 0,Y 677.254,Z 1006.515,A -85,B 0,C 180,E1 30654.063,E2 30654.063} C_VEL
LIN {X 0,Y 678.506,Z 986.245,A -85,B 0,C 180,E1 30653.143,E2 30653.143} C_VEL
LIN {X 0,Y 679.771,Z 964.183,A -85,B 0,C 180,E1 30652.271,E2 30652.271} C_VEL
LIN {X 0,Y 681.188,Z 936.023,A -85,B 0,C 180,E1 30651.341,E2 30651.341} C_VEL
LIN {X 0,Y 682.222,Z 911.41,A -85,B 0,C 180,E1 30650.697,E2 30650.697} C_VEL
LIN {X 0,Y 683.114,Z 886.167,A -85,B 0,C 180,E1 30650.18,E2 30650.18} C_VEL
LIN {X 0,Y 683.816,Z 852.477,A -85,B 0,C 180,E1 30649.7,E2 30649.7} C_VEL
LIN {X 0,Y 686.641,Z 629.501,A -85,B 0,C 180,E1 30646.845,E2 30646.845} C_VEL
LIN {X 0,Y 689.281,Z 434.641,A -85,B 0,C 180,E1 30644.271,E2 30644.271} C_VEL
LIN {X 0,Y 677.486,Z 417.171,A -85,B 0,C 180,E1 30642.975,E2 30642.975} C_VEL
LIN {X 0,Y 671.545,Z 408.991,A -85,B 0,C 180,E1 30642.299,E2 30642.299} C_VEL
LIN {X 0,Y 668.804,Z 405.147,A -85,B 0,C 180,E1 30641.978,E2 30641.978} C_VEL
LIN {X 0,Y 667.835,Z 403.905,A -85,B 0,C 180,E1 30641.866,E2 30641.866} C_VEL
LIN {X 0,Y 665.513,Z 401.21,A -85,B 0,C 180,E1 30641.597,E2 30641.597} C_VEL
LIN {X 0,Y 664.646,Z 398.443,A -85,B 0,C 180,E1 30641.448,E2 30641.448} C_VEL
LIN {X 0,Y 664.645,Z 398.439,A -85,B 0,C 180,E1 30638.25,E2 30638.25} C_VEL
LIN {X 0,Y 664.64,Z 398.42,A -85,B 0,C 180,E1 30635.073,E2 30635.073} C_VEL
LIN {X 0,Y 664.641,Z 398.437,A -85,B 0,C 180,E1 30631.951,E2 30631.951} C_VEL
LIN {X 0,Y 664.648,Z 398.431,A -85,B 0,C 180,E1 30628.876,E2 30628.876} C_VEL
LIN {X 0,Y 664.635,Z 398.415,A -85,B 0,C 180,E1 30625.689,E2 30625.689} C_VEL
LIN {X 0,Y 664.643,Z 398.439,A -85,B 0,C 180,E1 30622.558,E2 30622.558} C_VEL
LIN {X 0,Y 664.631,Z 398.422,A -85,B 0,C 180,E1 30619.419,E2 30619.419} C_VEL
LIN {X 0,Y 664.642,Z 398.429,A -85,B 0,C 180,E1 30616.339,E2 30616.339} C_VEL
LIN {X 0,Y 664.631,Z 398.429,A -85,B 0,C 180,E1 30613.219,E2 30613.219} C_VEL
LIN {X 0,Y 664.641,Z 398.423,A -85,B 0,C 180,E1 30610.138,E2 30610.138} C_VEL
LIN {X 0,Y 664.629,Z 398.431,A -85,B 0,C 180,E1 30606.999,E2 30606.999} C_VEL
LIN {X 0,Y 664.64,Z 398.422,A -85,B 0,C 180,E1 30603.968,E2 30603.968} C_VEL
LIN {X 0,Y 664.627,Z 398.432,A -85,B 0,C 180,E1 30600.776,E2 30600.776} C_VEL
LIN {X 0,Y 664.64,Z 398.42,A -85,B 0,C 180,E1 30597.758,E2 30597.758} C_VEL
LIN {X 0,Y 664.625,Z 398.433,A -85,B 0,C 180,E1 30594.561,E2 30594.561} C_VEL
LIN {X 0,Y 664.641,Z 398.418,A -85,B 0,C 180,E1 30591.522,E2 30591.522} C_VEL
LIN {X 0,Y 664.625,Z 398.435,A -85,B 0,C 180,E1 30588.351,E2 30588.351} C_VEL
LIN {X 0,Y 664.646,Z 398.416,A -85,B 0,C 180,E1 30585.271,E2 30585.271} C_VEL
LIN {X 0,Y 664.622,Z 398.437,A -85,B 0,C 180,E1 30582.127,E2 30582.127} C_VEL
LIN {X 0,Y 664.638,Z 398.419,A -85,B 0,C 180,E1 30579.108,E2 30579.108} C_VEL
LIN {X 0,Y 664.623,Z 398.431,A -85,B 0,C 180,E1 30575.939,E2 30575.939} C_VEL
LIN {X 0,Y 664.637,Z 398.439,A -85,B 0,C 180,E1 30572.881,E2 30572.881} C_VEL
LIN {X 0,Y 664.62,Z 398.423,A -85,B 0,C 180,E1 30569.72,E2 30569.72} C_VEL
LIN {X 0,Y 664.625,Z 398.426,A -85,B 0,C 180,E1 30566.771,E2 30566.771} C_VEL
LIN {X 0,Y 664.622,Z 398.436,A -85,B 0,C 180,E1 30563.54,E2 30563.54} C_VEL
LIN {X 0,Y 664.621,Z 398.558,A -85,B 0,C 180,E1 30560.829,E2 30560.829} C_VEL
LIN {X 0,Y 665.791,Z 401.696,A -85,B 0,C 180,E1 30560.449,E2 30560.449} C_VEL
LIN {X 0,Y 666.866,Z 403.525,A -85,B 0,C 180,E1 30560.19,E2 30560.19} C_VEL
LIN {X 0,Y 675.599,Z 421.838,A -85,B 0,C 180,E1 30557.899,E2 30557.899} C_VEL
LIN {X 0,Y 678.759,Z 428.163,A -85,B 0,C 180,E1 30557.154,E2 30557.154} C_VEL
LIN {X 0,Y 685.836,Z 439.034,A -85,B 0,C 180,E1 30556.359,E2 30556.359} C_VEL
LIN {X 0,Y 689.468,Z 454.297,A -85,B 0,C 180,E1 30555.819,E2 30555.819} C_VEL
LIN {X 0,Y 686.583,Z 663.708,A -85,B 0,C 180,E1 30553.055,E2 30553.055} C_VEL
LIN {X 0,Y 683.737,Z 888.809,A -85,B 0,C 180,E1 30550.175,E2 30550.175} C_VEL
LIN {X 0,Y 683.047,Z 918.117,A -85,B 0,C 180,E1 30549.738,E2 30549.738} C_VEL
LIN {X 0,Y 682.186,Z 942.311,A -85,B 0,C 180,E1 30549.237,E2 30549.237} C_VEL
LIN {X 0,Y 681.108,Z 967.849,A -85,B 0,C 180,E1 30548.561,E2 30548.561} C_VEL
LIN {X 0,Y 679.74,Z 994.866,A -85,B 0,C 180,E1 30547.658,E2 30547.658} C_VEL
LIN {X 0,Y 678.496,Z 1016.411,A -85,B 0,C 180,E1 30546.804,E2 30546.804} C_VEL
LIN {X 0,Y 677.246,Z 1036.654,A -85,B 0,C 180,E1 30545.885,E2 30545.885} C_VEL
LIN {X 0,Y 675.886,Z 1057.552,A -85,B 0,C 180,E1 30544.809,E2 30544.809} C_VEL
LIN {X 0,Y 674.177,Z 1082.619,A -85,B 0,C 180,E1 30543.335,E2 30543.335} C_VEL
LIN {X 0,Y 672.657,Z 1103.635,A -85,B 0,C 180,E1 30541.92,E2 30541.92} C_VEL
LIN {X 0,Y 671.371,Z 1122.226,A -85,B 0,C 180,E1 30540.524,E2 30540.524} C_VEL
LIN {X 0,Y 669.988,Z 1143.166,A -85,B 0,C 180,E1 30538.773,E2 30538.773} C_VEL
LIN {X 0,Y 668.649,Z 1162.423,A -85,B 0,C 180,E1 30536.946,E2 30536.946} C_VEL
LIN {X 0,Y 667.66,Z 1178.359,A -85,B 0,C 180,E1 30535.268,E2 30535.268} C_VEL
LIN {X 0,Y 666.62,Z 1196.402,A -85,B 0,C 180,E1 30533.143,E2 30533.143} C_VEL
LIN {X 0,Y 665.856,Z 1211.17,A -85,B 0,C 180,E1 30531.166,E2 30531.166} C_VEL
LIN {X 0,Y 665.303,Z 1223.671,A -85,B 0,C 180,E1 30529.295,E2 30529.295} C_VEL
LIN {X 0,Y 664.756,Z 1237.331,A -85,B 0,C 180,E1 30526.969,E2 30526.969} C_VEL
LIN {X 0,Y 664.422,Z 1248.057,A -85,B 0,C 180,E1 30524.826,E2 30524.826} C_VEL
LIN {X 0,Y 664.21,Z 1256.498,A -85,B 0,C 180,E1 30522.877,E2 30522.877} C_VEL
LIN {X 0,Y 664.046,Z 1263.651,A -85,B 0,C 180,E1 30520.94,E2 30520.94} C_VEL
LIN {X 0,Y 663.974,Z 1270.585,A -85,B 0,C 180,E1 30518.665,E2 30518.665} C_VEL
LIN {X 0,Y 663.936,Z 1275.961,A -85,B 0,C 180,E1 30516.297,E2 30516.297} C_VEL
LIN {X 0,Y 663.918,Z 1279.477,A -85,B 0,C 180,E1 30514.063,E2 30514.063} C_VEL
LIN {X 0,Y 663.91,Z 1281.6,A -85,B 0,C 180,E1 30511.557,E2 30511.557} C_VEL
LIN {X 0,Y 663.867,Z 1281.873,A -85,B 0,C 180,E1 30509.486,E2 30509.486} C_VEL
LIN {X 0,Y 663.906,Z 1281.017,A -85,B 0,C 180,E1 30507.587,E2 30507.587} C_VEL
LIN {X 0,Y 663.914,Z 1278.994,A -85,B 0,C 180,E1 30505.57,E2 30505.57} C_VEL
LIN {X 0,Y 663.931,Z 1275.087,A -85,B 0,C 180,E1 30503.258,E2 30503.258} C_VEL
LIN {X 0,Y 663.947,Z 1269.597,A -85,B 0,C 180,E1 30500.994,E2 30500.994} C_VEL
LIN {X 0,Y 664.051,Z 1263.373,A -85,B 0,C 180,E1 30498.98,E2 30498.98} C_VEL
LIN {X 0,Y 664.214,Z 1256.172,A -85,B 0,C 180,E1 30497.043,E2 30497.043} C_VEL
LIN {X 0,Y 664.43,Z 1247.685,A -85,B 0,C 180,E1 30495.093,E2 30495.093} C_VEL
LIN {X 0,Y 664.823,Z 1235.825,A -85,B 0,C 180,E1 30492.754,E2 30492.754} C_VEL
LIN {X 0,Y 665.328,Z 1223.048,A -85,B 0,C 180,E1 30490.607,E2 30490.607} C_VEL
LIN {X 0,Y 665.907,Z 1210.21,A -85,B 0,C 180,E1 30488.698,E2 30488.698} C_VEL
LIN {X 0,Y 666.756,Z 1194.298,A -85,B 0,C 180,E1 30486.59,E2 30486.59} C_VEL
LIN {X 0,Y 667.697,Z 1177.591,A -85,B 0,C 180,E1 30484.647,E2 30484.647} C_VEL
LIN {X 0,Y 668.708,Z 1161.577,A -85,B 0,C 180,E1 30482.97,E2 30482.97} C_VEL
LIN {X 0,Y 670.086,Z 1141.656,A -85,B 0,C 180,E1 30481.094,E2 30481.094} C_VEL
LIN {X 0,Y 671.43,Z 1121.282,A -85,B 0,C 180,E1 30479.402,E2 30479.402} C_VEL
LIN {X 0,Y 672.73,Z 1102.653,A -85,B 0,C 180,E1 30478.01,E2 30478.01} C_VEL
LIN {X 0,Y 674.452,Z 1078.965,A -85,B 0,C 180,E1 30476.435,E2 30476.435} C_VEL
LIN {X 0,Y 676.001,Z 1055.659,A -85,B 0,C 180,E1 30475.088,E2 30475.088} C_VEL
LIN {X 0,Y 677.352,Z 1034.83,A -85,B 0,C 180,E1 30474.026,E2 30474.026} C_VEL
LIN {X 0,Y 678.894,Z 1009.837,A -85,B 0,C 180,E1 30472.914,E2 30472.914} C_VEL
LIN {X 0,Y 680.291,Z 983.665,A -85,B 0,C 180,E1 30471.946,E2 30471.946} C_VEL
LIN {X 0,Y 681.417,Z 960.73,A -85,B 0,C 180,E1 30471.237,E2 30471.237} C_VEL
LIN {X 0,Y 682.463,Z 935.511,A -85,B 0,C 180,E1 30470.605,E2 30470.605} C_VEL
LIN {X 0,Y 683.373,Z 906.736,A -85,B 0,C 180,E1 30470.072,E2 30470.072} C_VEL
LIN {X 0,Y 684.834,Z 799.599,A -85,B 0,C 180,E1 30468.694,E2 30468.694} C_VEL
LIN {X 0,Y 687.686,Z 581.744,A -85,B 0,C 180,E1 30465.873,E2 30465.873} C_VEL
LIN {X 0,Y 689.361,Z 453.068,A -85,B 0,C 180,E1 30464.154,E2 30464.154} C_VEL
LIN {X 0,Y 685.406,Z 438.053,A -85,B 0,C 180,E1 30463.589,E2 30463.589} C_VEL
LIN {X 0,Y 678.25,Z 427.36,A -85,B 0,C 180,E1 30462.773,E2 30462.773} C_VEL
LIN {X 0,Y 670.129,Z 410.499,A -85,B 0,C 180,E1 30460.696,E2 30460.696} C_VEL
LIN {X 0,Y 666.167,Z 402.26,A -85,B 0,C 180,E1 30459.636,E2 30459.636} C_VEL
LIN {X 0,Y 664.719,Z 399.189,A -85,B 0,C 180,E1 30459.235,E2 30459.235} C_VEL
LIN {X 0,Y 664.589,Z 398.449,A -85,B 0,C 180,E1 30459.135,E2 30459.135} C_VEL
LIN {X 0,Y 664.639,Z 398.435,A -85,B 0,C 180,E1 30456.245,E2 30456.245} C_VEL
LIN {X 0,Y 664.585,Z 398.432,A -85,B 0,C 180,E1 30453.206,E2 30453.206} C_VEL
LIN {X 0,Y 664.583,Z 398.434,A -85,B 0,C 180,E1 30450.566,E2 30450.566} C_VEL
LIN {X 0,Y 664.628,Z 398.444,A -85,B 0,C 180,E1 30447.507,E2 30447.507} C_VEL
LIN {X 0,Y 664.562,Z 398.431,A -85,B 0,C 180,E1 30444.681,E2 30444.681} C_VEL
LIN {X 0,Y 664.617,Z 398.443,A -85,B 0,C 180,E1 30441.907,E2 30441.907} C_VEL
LIN {X 0,Y 664.568,Z 398.444,A -85,B 0,C 180,E1 30438.871,E2 30438.871} C_VEL
LIN {X 0,Y 664.554,Z 398.442,A -85,B 0,C 180,E1 30436.342,E2 30436.342} C_VEL
LIN {X 0,Y 664.634,Z 398.426,A -85,B 0,C 180,E1 30433.485,E2 30433.485} C_VEL
LIN {X 0,Y 664.547,Z 398.438,A -85,B 0,C 180,E1 30430.577,E2 30430.577} C_VEL
LIN {X 0,Y 664.541,Z 398.433,A -85,B 0,C 180,E1 30428.044,E2 30428.044} C_VEL
LIN {X 0,Y 664.623,Z 398.436,A -85,B 0,C 180,E1 30425.092,E2 30425.092} C_VEL
LIN {X 0,Y 664.545,Z 398.433,A -85,B 0,C 180,E1 30422.242,E2 30422.242} C_VEL
LIN {X 0,Y 664.559,Z 398.447,A -85,B 0,C 180,E1 30419.741,E2 30419.741} C_VEL
LIN {X 0,Y 664.613,Z 398.419,A -85,B 0,C 180,E1 30416.723,E2 30416.723} C_VEL
LIN {X 0,Y 664.56,Z 398.445,A -85,B 0,C 180,E1 30413.936,E2 30413.936} C_VEL
LIN {X 0,Y 664.586,Z 398.424,A -85,B 0,C 180,E1 30411.347,E2 30411.347} C_VEL
LIN {X 0,Y 664.59,Z 398.443,A -85,B 0,C 180,E1 30408.193,E2 30408.193} C_VEL
LIN {X 0,Y 664.573,Z 398.427,A -85,B 0,C 180,E1 30405.537,E2 30405.537} C_VEL
LIN {X 0,Y 664.653,Z 398.441,A -85,B 0,C 180,E1 30402.58,E2 30402.58} C_VEL
LIN {X 0,Y 664.58,Z 398.42,A -85,B 0,C 180,E1 30399.588,E2 30399.588} C_VEL
LIN {X 0,Y 664.633,Z 398.445,A -85,B 0,C 180,E1 30396.786,E2 30396.786} C_VEL
LIN {X 0,Y 664.598,Z 398.429,A -85,B 0,C 180,E1 30393.651,E2 30393.651} C_VEL
LIN {X 0,Y 664.618,Z 398.434,A -85,B 0,C 180,E1 30390.827,E2 30390.827} C_VEL
LIN {X 0,Y 664.616,Z 398.441,A -85,B 0,C 180,E1 30387.616,E2 30387.616} C_VEL
LIN {X 0,Y 664.618,Z 398.423,A -85,B 0,C 180,E1 30384.71,E2 30384.71} C_VEL
LIN {X 0,Y 664.613,Z 398.443,A -85,B 0,C 180,E1 30383.384,E2 30383.384} C_VEL
LIN {X 0,Y 663.601,Z 398.566,A -85,B 0,C 180,E1 30382.72,E2 30382.72} C_VEL
LIN {X 0,Y 657.214,Z 399.346,A -85,B 0,C 180,E1 30380.858,E2 30380.858} C_VEL
LIN {X 0,Y 656.707,Z 399.418,A -85,B 0,C 180,E1 30380.374,E2 30380.374} C_VEL
LIN {X 0,Y 656.706,Z 399.644,A -85,B 0,C 180,E1 30379.217,E2 30379.217} C_VEL
LIN {X 0,Y 657.922,Z 402.829,A -85,B 0,C 180,E1 30379.041,E2 30379.041} C_VEL
LIN {X 0,Y 660.852,Z 405.992,A -85,B 0,C 180,E1 30378.695,E2 30378.695} C_VEL
LIN {X 0,Y 663.464,Z 409.809,A -85,B 0,C 180,E1 30378.375,E2 30378.375} C_VEL
LIN {X 0,Y 665.098,Z 411.831,A -85,B 0,C 180,E1 30378.183,E2 30378.183} C_VEL
LIN {X 0,Y 675.025,Z 425.489,A -85,B 0,C 180,E1 30377.032,E2 30377.032} C_VEL
LIN {X 0,Y 683.656,Z 438.575,A -85,B 0,C 180,E1 30376.065,E2 30376.065} C_VEL
LIN {X 0,Y 680.594,Z 643.401,A -85,B 0,C 180,E1 30373.345,E2 30373.345} C_VEL
LIN {X 0,Y 677.411,Z 869.032,A -85,B 0,C 180,E1 30370.43,E2 30370.43} C_VEL
LIN {X 0,Y 676.691,Z 892.951,A -85,B 0,C 180,E1 30370.039,E2 30370.039} C_VEL
LIN {X 0,Y 675.69,Z 918.743,A -85,B 0,C 180,E1 30369.472,E2 30369.472} C_VEL
LIN {X 0,Y 674.344,Z 945.648,A -85,B 0,C 180,E1 30368.7,E2 30368.7} C_VEL
LIN {X 0,Y 673.129,Z 967.396,A -85,B 0,C 180,E1 30367.942,E2 30367.942} C_VEL
LIN {X 0,Y 671.84,Z 987.927,A -85,B 0,C 180,E1 30367.113,E2 30367.113} C_VEL
LIN {X 0,Y 670.424,Z 1008.986,A -85,B 0,C 180,E1 30366.14,E2 30366.14} C_VEL
LIN {X 0,Y 668.659,Z 1033.888,A -85,B 0,C 180,E1 30364.819,E2 30364.819} C_VEL
LIN {X 0,Y 666.893,Z 1056.511,A -85,B 0,C 180,E1 30363.429,E2 30363.429} C_VEL
LIN {X 0,Y 665.377,Z 1076.125,A -85,B 0,C 180,E1 30362.076,E2 30362.076} C_VEL
LIN {X 0,Y 663.779,Z 1097.836,A -85,B 0,C 180,E1 30360.4,E2 30360.4} C_VEL
LIN {X 0,Y 662.2,Z 1118.381,A -85,B 0,C 180,E1 30358.591,E2 30358.591} C_VEL
LIN {X 0,Y 660.996,Z 1134.864,A -85,B 0,C 180,E1 30356.982,E2 30356.982} C_VEL
LIN {X 0,Y 659.81,Z 1153.073,A -85,B 0,C 180,E1 30355.006,E2 30355.006} C_VEL
LIN {X 0,Y 658.715,Z 1169.683,A -85,B 0,C 180,E1 30352.956,E2 30352.956} C_VEL
LIN {X 0,Y 657.964,Z 1183.29,A -85,B 0,C 180,E1 30351.079,E2 30351.079} C_VEL
LIN {X 0,Y 657.27,Z 1197.871,A -85,B 0,C 180,E1 30348.809,E2 30348.809} C_VEL
LIN {X 0,Y 656.729,Z 1209.94,A -85,B 0,C 180,E1 30346.628,E2 30346.628} C_VEL
LIN {X 0,Y 656.448,Z 1219.223,A -85,B 0,C 180,E1 30344.709,E2 30344.709} C_VEL
LIN {X 0,Y 656.212,Z 1227.771,A -85,B 0,C 180,E1 30342.67,E2 30342.67} C_VEL
LIN {X 0,Y 656.045,Z 1236.4,A -85,B 0,C 180,E1 30340.179,E2 30340.179} C_VEL
LIN {X 0,Y 655.936,Z 1242.444,A -85,B 0,C 180,E1 30337.969,E2 30337.969} C_VEL
LIN {X 0,Y 655.927,Z 1246.972,A -85,B 0,C 180,E1 30335.77,E2 30335.77} C_VEL
LIN {X 0,Y 655.912,Z 1250.236,A -85,B 0,C 180,E1 30333.404,E2 30333.404} C_VEL
LIN {X 0,Y 655.888,Z 1251.704,A -85,B 0,C 180,E1 30331.132,E2 30331.132} C_VEL
LIN {X 0,Y 655.864,Z 1251.837,A -85,B 0,C 180,E1 30329.297,E2 30329.297} C_VEL
LIN {X 0,Y 655.904,Z 1250.979,A -85,B 0,C 180,E1 30327.462,E2 30327.462} C_VEL
LIN {X 0,Y 655.912,Z 1248.964,A -85,B 0,C 180,E1 30325.45,E2 30325.45} C_VEL
LIN {X 0,Y 655.934,Z 1244.988,A -85,B 0,C 180,E1 30323.08,E2 30323.08} C_VEL
LIN {X 0,Y 655.95,Z 1239.703,A -85,B 0,C 180,E1 30320.875,E2 30320.875} C_VEL
LIN {X 0,Y 656.068,Z 1233.5,A -85,B 0,C 180,E1 30318.836,E2 30318.836} C_VEL
LIN {X 0,Y 656.239,Z 1226.321,A -85,B 0,C 180,E1 30316.875,E2 30316.875} C_VEL
LIN {X 0,Y 656.471,Z 1218.051,A -85,B 0,C 180,E1 30314.943,E2 30314.943} C_VEL
LIN {X 0,Y 656.88,Z 1207.096,A -85,B 0,C 180,E1 30312.73,E2 30312.73} C_VEL
LIN {X 0,Y 657.451,Z 1193.848,A -85,B 0,C 180,E1 30310.449,E2 30310.449} C_VEL
LIN {X 0,Y 658.087,Z 1181.108,A -85,B 0,C 180,E1 30308.517,E2 30308.517} C_VEL
LIN {X 0,Y 659.014,Z 1165.32,A -85,B 0,C 180,E1 30306.384,E2 30306.384} C_VEL
LIN {X 0,Y 660.087,Z 1147.907,A -85,B 0,C 180,E1 30304.325,E2 30304.325} C_VEL
LIN {X 0,Y 661.22,Z 1131.922,A -85,B 0,C 180,E1 30302.629,E2 30302.629} C_VEL
LIN {X 0,Y 662.709,Z 1112.058,A -85,B 0,C 180,E1 30300.732,E2 30300.732} C_VEL
LIN {X 0,Y 664.201,Z 1091.558,A -85,B 0,C 180,E1 30299.01,E2 30299.01} C_VEL
LIN {X 0,Y 665.659,Z 1072.668,A -85,B 0,C 180,E1 30297.585,E2 30297.585} C_VEL
LIN {X 0,Y 667.493,Z 1049.526,A -85,B 0,C 180,E1 30296.028,E2 30296.028} C_VEL
LIN {X 0,Y 669.173,Z 1026.265,A -85,B 0,C 180,E1 30294.669,E2 30294.669} C_VEL
LIN {X 0,Y 670.639,Z 1005.493,A -85,B 0,C 180,E1 30293.599,E2 30293.599} C_VEL
LIN {X 0,Y 672.151,Z 982.836,A -85,B 0,C 180,E1 30292.576,E2 30292.576} C_VEL
LIN {X 0,Y 673.817,Z 955.203,A -85,B 0,C 180,E1 30291.526,E2 30291.526} C_VEL
LIN {X 0,Y 675.052,Z 931.928,A -85,B 0,C 180,E1 30290.796,E2 30290.796} C_VEL
LIN {X 0,Y 676.125,Z 908.127,A -85,B 0,C 180,E1 30290.187,E2 30290.187} C_VEL
LIN {X 0,Y 677.136,Z 880.251,A -85,B 0,C 180,E1 30289.644,E2 30289.644} C_VEL
LIN {X 0,Y 677.981,Z 831.65,A -85,B 0,C 180,E1 30288.996,E2 30288.996} C_VEL
LIN {X 0,Y 681.084,Z 610.099,A -85,B 0,C 180,E1 30286.129,E2 30286.129} C_VEL
LIN {X 0,Y 683.627,Z 438.342,A -85,B 0,C 180,E1 30283.839,E2 30283.839} C_VEL
LIN {X 0,Y 671.511,Z 420.477,A -85,B 0,C 180,E1 30282.475,E2 30282.475} C_VEL
LIN {X 0,Y 664.618,Z 410.959,A -85,B 0,C 180,E1 30281.666,E2 30281.666} C_VEL
LIN {X 0,Y 661.425,Z 407.117,A -85,B 0,C 180,E1 30281.29,E2 30281.29} C_VEL
LIN {X 0,Y 660.138,Z 405.061,A -85,B 0,C 180,E1 30281.128,E2 30281.128} C_VEL
LIN {X 0,Y 657.618,Z 402.298,A -85,B 0,C 180,E1 30280.829,E2 30280.829} C_VEL
LIN {X 0,Y 656.695,Z 399.433,A -85,B 0,C 180,E1 30280.668,E2 30280.668} C_VEL
LIN {X 0,Y 656.691,Z 399.428,A -85,B 0,C 180,E1 30277.631,E2 30277.631} C_VEL
LIN {X 0,Y 656.688,Z 399.406,A -85,B 0,C 180,E1 30274.607,E2 30274.607} C_VEL
LIN {X 0,Y 656.688,Z 399.426,A -85,B 0,C 180,E1 30271.587,E2 30271.587} C_VEL
LIN {X 0,Y 656.693,Z 399.43,A -85,B 0,C 180,E1 30268.562,E2 30268.562} C_VEL
LIN {X 0,Y 656.687,Z 399.402,A -85,B 0,C 180,E1 30265.525,E2 30265.525} C_VEL
LIN {X 0,Y 656.698,Z 399.426,A -85,B 0,C 180,E1 30262.447,E2 30262.447} C_VEL
LIN {X 0,Y 656.69,Z 399.411,A -85,B 0,C 180,E1 30259.386,E2 30259.386} C_VEL
LIN {X 0,Y 656.703,Z 399.417,A -85,B 0,C 180,E1 30256.361,E2 30256.361} C_VEL
LIN {X 0,Y 656.691,Z 399.417,A -85,B 0,C 180,E1 30253.203,E2 30253.203} C_VEL
LIN {X 0,Y 656.701,Z 399.409,A -85,B 0,C 180,E1 30250.084,E2 30250.084} C_VEL
LIN {X 0,Y 656.69,Z 399.42,A -85,B 0,C 180,E1 30246.997,E2 30246.997} C_VEL
LIN {X 0,Y 656.701,Z 399.408,A -85,B 0,C 180,E1 30243.929,E2 30243.929} C_VEL
LIN {X 0,Y 656.689,Z 399.421,A -85,B 0,C 180,E1 30240.785,E2 30240.785} C_VEL
LIN {X 0,Y 656.701,Z 399.406,A -85,B 0,C 180,E1 30237.731,E2 30237.731} C_VEL
LIN {X 0,Y 656.688,Z 399.422,A -85,B 0,C 180,E1 30234.583,E2 30234.583} C_VEL
LIN {X 0,Y 656.703,Z 399.404,A -85,B 0,C 180,E1 30231.507,E2 30231.507} C_VEL
LIN {X 0,Y 656.684,Z 399.425,A -85,B 0,C 180,E1 30228.316,E2 30228.316} C_VEL
LIN {X 0,Y 656.708,Z 399.403,A -85,B 0,C 180,E1 30225.27,E2 30225.27} C_VEL
LIN {X 0,Y 656.682,Z 399.427,A -85,B 0,C 180,E1 30222.087,E2 30222.087} C_VEL
LIN {X 0,Y 656.703,Z 399.407,A -85,B 0,C 180,E1 30219.034,E2 30219.034} C_VEL
LIN {X 0,Y 656.682,Z 399.42,A -85,B 0,C 180,E1 30215.916,E2 30215.916} C_VEL
LIN {X 0,Y 656.695,Z 399.427,A -85,B 0,C 180,E1 30212.918,E2 30212.918} C_VEL
LIN {X 0,Y 656.679,Z 399.41,A -85,B 0,C 180,E1 30209.696,E2 30209.696} C_VEL
LIN {X 0,Y 656.691,Z 399.411,A -85,B 0,C 180,E1 30206.714,E2 30206.714} C_VEL
LIN {X 0,Y 656.68,Z 399.422,A -85,B 0,C 180,E1 30203.512,E2 30203.512} C_VEL
LIN {X 0,Y 656.713,Z 399.572,A -85,B 0,C 180,E1 30201.561,E2 30201.561} C_VEL
LIN {X 0,Y 658.03,Z 403.003,A -85,B 0,C 180,E1 30201.129,E2 30201.129} C_VEL
LIN {X 0,Y 659.181,Z 405.274,A -85,B 0,C 180,E1 30200.818,E2 30200.818} C_VEL
LIN {X 0,Y 663.29,Z 413.68,A -85,B 0,C 180,E1 30199.706,E2 30199.706} C_VEL
LIN {X 0,Y 670.162,Z 427.825,A -85,B 0,C 180,E1 30197.954,E2 30197.954} C_VEL
LIN {X 0,Y 680.835,Z 443.544,A -85,B 0,C 180,E1 30196.734,E2 30196.734} C_VEL
LIN {X 0,Y 683.853,Z 456.442,A -85,B 0,C 180,E1 30196.273,E2 30196.273} C_VEL
LIN {X 0,Y 680.707,Z 665.505,A -85,B 0,C 180,E1 30193.494,E2 30193.494} C_VEL
LIN {X 0,Y 677.598,Z 890.591,A -85,B 0,C 180,E1 30190.59,E2 30190.59} C_VEL
LIN {X 0,Y 676.845,Z 918.904,A -85,B 0,C 180,E1 30190.159,E2 30190.159} C_VEL
LIN {X 0,Y 675.93,Z 942.682,A -85,B 0,C 180,E1 30189.661,E2 30189.661} C_VEL
LIN {X 0,Y 674.757,Z 968.261,A -85,B 0,C 180,E1 30188.979,E2 30188.979} C_VEL
LIN {X 0,Y 673.277,Z 994.869,A -85,B 0,C 180,E1 30188.084,E2 30188.084} C_VEL
LIN {X 0,Y 671.904,Z 1016.797,A -85,B 0,C 180,E1 30187.208,E2 30187.208} C_VEL
LIN {X 0,Y 670.506,Z 1037.656,A -85,B 0,C 180,E1 30186.25,E2 30186.25} C_VEL
LIN {X 0,Y 668.877,Z 1060.842,A -85,B 0,C 180,E1 30185.034,E2 30185.034} C_VEL
LIN {X 0,Y 666.981,Z 1085.531,A -85,B 0,C 180,E1 30183.538,E2 30183.538} C_VEL
LIN {X 0,Y 665.456,Z 1105.136,A -85,B 0,C 180,E1 30182.193,E2 30182.193} C_VEL
LIN {X 0,Y 663.952,Z 1125.19,A -85,B 0,C 180,E1 30180.656,E2 30180.656} C_VEL
LIN {X 0,Y 662.315,Z 1147.038,A -85,B 0,C 180,E1 30178.761,E2 30178.761} C_VEL
LIN {X 0,Y 661.07,Z 1163.819,A -85,B 0,C 180,E1 30177.134,E2 30177.134} C_VEL
LIN {X 0,Y 659.902,Z 1181.474,A -85,B 0,C 180,E1 30175.232,E2 30175.232} C_VEL
LIN {X 0,Y 658.762,Z 1198.911,A -85,B 0,C 180,E1 30173.102,E2 30173.102} C_VEL
LIN {X 0,Y 658.032,Z 1212.087,A -85,B 0,C 180,E1 30171.298,E2 30171.298} C_VEL
LIN {X 0,Y 657.388,Z 1225.289,A -85,B 0,C 180,E1 30169.275,E2 30169.275} C_VEL
LIN {X 0,Y 656.789,Z 1238.729,A -85,B 0,C 180,E1 30166.908,E2 30166.908} C_VEL
LIN {X 0,Y 656.467,Z 1248.469,A -85,B 0,C 180,E1 30164.92,E2 30164.92} C_VEL
LIN {X 0,Y 656.235,Z 1256.856,A -85,B 0,C 180,E1 30162.946,E2 30162.946} C_VEL
LIN {X 0,Y 656.054,Z 1264.559,A -85,B 0,C 180,E1 30160.808,E2 30160.808} C_VEL
LIN {X 0,Y 655.962,Z 1271.904,A -85,B 0,C 180,E1 30158.242,E2 30158.242} C_VEL
LIN {X 0,Y 655.931,Z 1276.563,A -85,B 0,C 180,E1 30156.041,E2 30156.041} C_VEL
LIN {X 0,Y 655.914,Z 1279.988,A -85,B 0,C 180,E1 30153.675,E2 30153.675} C_VEL
LIN {X 0,Y 655.899,Z 1281.668,A -85,B 0,C 180,E1 30151.314,E2 30151.314} C_VEL
LIN {X 0,Y 655.864,Z 1281.85,A -85,B 0,C 180,E1 30149.393,E2 30149.393} C_VEL
LIN {X 0,Y 655.906,Z 1281.017,A -85,B 0,C 180,E1 30147.558,E2 30147.558} C_VEL
LIN {X 0,Y 655.914,Z 1279.028,A -85,B 0,C 180,E1 30145.544,E2 30145.544} C_VEL
LIN {X 0,Y 655.933,Z 1275.259,A -85,B 0,C 180,E1 30143.264,E2 30143.264} C_VEL
LIN {X 0,Y 655.953,Z 1269.851,A -85,B 0,C 180,E1 30140.971,E2 30140.971} C_VEL
LIN {X 0,Y 656.073,Z 1263.374,A -85,B 0,C 180,E1 30138.844,E2 30138.844} C_VEL
LIN {X 0,Y 656.239,Z 1256.53,A -85,B 0,C 180,E1 30136.972,E2 30136.972} C_VEL
LIN {X 0,Y 656.473,Z 1248.097,A -85,B 0,C 180,E1 30134.998,E2 30134.998} C_VEL
LIN {X 0,Y 656.888,Z 1236.912,A -85,B 0,C 180,E1 30132.738,E2 30132.738} C_VEL
LIN {X 0,Y 657.462,Z 1223.624,A -85,B 0,C 180,E1 30130.458,E2 30130.458} C_VEL
LIN {X 0,Y 658.1,Z 1210.857,A -85,B 0,C 180,E1 30128.526,E2 30128.526} C_VEL
LIN {X 0,Y 659.033,Z 1195.047,A -85,B 0,C 180,E1 30126.394,E2 30126.394} C_VEL
LIN {X 0,Y 660.112,Z 1177.509,A -85,B 0,C 180,E1 30124.325,E2 30124.325} C_VEL
LIN {X 0,Y 661.247,Z 1161.578,A -85,B 0,C 180,E1 30122.639,E2 30122.639} C_VEL
LIN {X 0,Y 662.735,Z 1141.656,A -85,B 0,C 180,E1 30120.743,E2 30120.743} C_VEL
LIN {X 0,Y 664.186,Z 1121.763,A -85,B 0,C 180,E1 30119.072,E2 30119.072} C_VEL
LIN {X 0,Y 665.603,Z 1103.318,A -85,B 0,C 180,E1 30117.677,E2 30117.677} C_VEL
LIN {X 0,Y 667.419,Z 1080.541,A -85,B 0,C 180,E1 30116.137,E2 30116.137} C_VEL
LIN {X 0,Y 669.152,Z 1056.552,A -85,B 0,C 180,E1 30114.73,E2 30114.73} C_VEL
LIN {X 0,Y 670.619,Z 1035.831,A -85,B 0,C 180,E1 30113.661,E2 30113.661} C_VEL
LIN {X 0,Y 672.125,Z 1013.225,A -85,B 0,C 180,E1 30112.637,E2 30112.637} C_VEL
LIN {X 0,Y 673.826,Z 984.988,A -85,B 0,C 180,E1 30111.563,E2 30111.563} C_VEL
LIN {X 0,Y 675.074,Z 961.473,A -85,B 0,C 180,E1 30110.828,E2 30110.828} C_VEL
LIN {X 0,Y 676.159,Z 937.331,A -85,B 0,C 180,E1 30110.214,E2 30110.214} C_VEL
LIN {X 0,Y 677.18,Z 908.856,A -85,B 0,C 180,E1 30109.667,E2 30109.667} C_VEL
LIN {X 0,Y 678.141,Z 849.474,A -85,B 0,C 180,E1 30108.885,E2 30108.885} C_VEL
LIN {X 0,Y 681.219,Z 630.25,A -85,B 0,C 180,E1 30106.043,E2 30106.043} C_VEL
LIN {X 0,Y 683.782,Z 455.362,A -85,B 0,C 180,E1 30103.704,E2 30103.704} C_VEL
LIN {X 0,Y 680.507,Z 442.912,A -85,B 0,C 180,E1 30103.227,E2 30103.227} C_VEL
LIN {X 0,Y 669.719,Z 427.078,A -85,B 0,C 180,E1 30101.978,E2 30101.978} C_VEL
LIN {X 0,Y 660.731,Z 408.088,A -85,B 0,C 180,E1 30099.576,E2 30099.576} C_VEL
LIN {X 0,Y 658.789,Z 404.083,A -85,B 0,C 180,E1 30099.041,E2 30099.041} C_VEL
LIN {X 0,Y 656.866,Z 400.424,A -85,B 0,C 180,E1 30098.528,E2 30098.528} C_VEL
LIN {X 0,Y 656.69,Z 399.415,A -85,B 0,C 180,E1 30098.406,E2 30098.406} C_VEL
LIN {X 0,Y 656.656,Z 399.431,A -85,B 0,C 180,E1 30095.309,E2 30095.309} C_VEL
LIN {X 0,Y 656.648,Z 399.429,A -85,B 0,C 180,E1 30092.619,E2 30092.619} C_VEL
LIN {X 0,Y 656.691,Z 399.407,A -85,B 0,C 180,E1 30089.56,E2 30089.56} C_VEL
LIN {X 0,Y 656.632,Z 399.431,A -85,B 0,C 180,E1 30086.791,E2 30086.791} C_VEL
LIN {X 0,Y 656.672,Z 399.418,A -85,B 0,C 180,E1 30083.988,E2 30083.988} C_VEL
LIN {X 0,Y 656.635,Z 399.414,A -85,B 0,C 180,E1 30080.968,E2 30080.968} C_VEL
LIN {X 0,Y 656.62,Z 399.432,A -85,B 0,C 180,E1 30078.374,E2 30078.374} C_VEL
LIN {X 0,Y 656.705,Z 399.405,A -85,B 0,C 180,E1 30075.453,E2 30075.453} C_VEL
LIN {X 0,Y 656.611,Z 399.436,A -85,B 0,C 180,E1 30072.578,E2 30072.578} C_VEL
LIN {X 0,Y 656.612,Z 399.423,A -85,B 0,C 180,E1 30069.997,E2 30069.997} C_VEL
LIN {X 0,Y 656.646,Z 399.437,A -85,B 0,C 180,E1 30066.909,E2 30066.909} C_VEL
LIN {X 0,Y 656.602,Z 399.424,A -85,B 0,C 180,E1 30064.192,E2 30064.192} C_VEL
LIN {X 0,Y 656.657,Z 399.422,A -85,B 0,C 180,E1 30061.396,E2 30061.396} C_VEL
LIN {X 0,Y 656.625,Z 399.421,A -85,B 0,C 180,E1 30058.342,E2 30058.342} C_VEL
LIN {X 0,Y 656.621,Z 399.421,A -85,B 0,C 180,E1 30055.721,E2 30055.721} C_VEL
LIN {X 0,Y 656.702,Z 399.418,A -85,B 0,C 180,E1 30052.74,E2 30052.74} C_VEL
LIN {X 0,Y 656.626,Z 399.42,A -85,B 0,C 180,E1 30049.826,E2 30049.826} C_VEL
LIN {X 0,Y 656.684,Z 399.427,A -85,B 0,C 180,E1 30046.997,E2 30046.997} C_VEL
LIN {X 0,Y 656.644,Z 399.423,A -85,B 0,C 180,E1 30043.911,E2 30043.911} C_VEL
LIN {X 0,Y 656.652,Z 399.434,A -85,B 0,C 180,E1 30041.259,E2 30041.259} C_VEL
LIN {X 0,Y 656.683,Z 399.426,A -85,B 0,C 180,E1 30038.096,E2 30038.096} C_VEL
LIN {X 0,Y 656.651,Z 399.421,A -85,B 0,C 180,E1 30035.244,E2 30035.244} C_VEL
LIN {X 0,Y 656.714,Z 399.428,A -85,B 0,C 180,E1 30032.189,E2 30032.189} C_VEL
LIN {X 0,Y 656.655,Z 399.408,A -85,B 0,C 180,E1 30029.227,E2 30029.227} C_VEL
LIN {X 0,Y 656.706,Z 399.41,A -85,B 0,C 180,E1 30026.238,E2 30026.238} C_VEL
LIN {X 0,Y 656.668,Z 399.434,A -85,B 0,C 180,E1 30023.207,E2 30023.207} C_VEL
LIN {X 0,Y 656.707,Z 399.418,A -85,B 0,C 180,E1 30020.374,E2 30020.374} C_VEL
LIN {X 0,Y 656.823,Z 400.244,A -85,B 0,C 180,E1 30020.008,E2 30020.008} C_VEL
LIN {X 0,Y 657.216,Z 402.923,A -85,B 0,C 180,E1 30019.596,E2 30019.596} C_VEL
LIN {X 0,Y 658.249,Z 408.341,A -85,B 0,C 180,E1 30019.112,E2 30019.112} C_VEL
LIN {X 0,Y 660.807,Z 416.569,A -85,B 0,C 180,E1 30018.557,E2 30018.557} C_VEL
LIN {X 0,Y 663.621,Z 421.344,A -85,B 0,C 180,E1 30018.176,E2 30018.176} C_VEL
LIN {X 0,Y 664.204,Z 422.006,A -85,B 0,C 180,E1 30018.108,E2 30018.108} C_VEL
LIN {X 0,Y 673.528,Z 435.427,A -85,B 0,C 180,E1 30017.017,E2 30017.017} C_VEL
LIN {X 0,Y 678.038,Z 442.597,A -85,B 0,C 180,E1 30016.5,E2 30016.5} C_VEL
LIN {X 0,Y 674.701,Z 648.282,A -85,B 0,C 180,E1 30013.75,E2 30013.75} C_VEL
LIN {X 0,Y 671.281,Z 870.327,A -85,B 0,C 180,E1 30010.856,E2 30010.856} C_VEL
LIN {X 0,Y 670.514,Z 893.886,A -85,B 0,C 180,E1 30010.464,E2 30010.464} C_VEL
LIN {X 0,Y 669.396,Z 920.493,A -85,B 0,C 180,E1 30009.868,E2 30009.868} C_VEL
LIN {X 0,Y 667.974,Z 946.403,A -85,B 0,C 180,E1 30009.112,E2 30009.112} C_VEL
LIN {X 0,Y 666.698,Z 967.41,A -85,B 0,C 180,E1 30008.374,E2 30008.374} C_VEL
LIN {X 0,Y 665.302,Z 987.937,A -85,B 0,C 180,E1 30007.541,E2 30007.541} C_VEL
LIN {X 0,Y 663.771,Z 1009.001,A -85,B 0,C 180,E1 30006.56,E2 30006.56} C_VEL
LIN {X 0,Y 661.885,Z 1033.741,A -85,B 0,C 180,E1 30005.238,E2 30005.238} C_VEL
LIN {X 0,Y 659.969,Z 1056.517,A -85,B 0,C 180,E1 30003.827,E2 30003.827} C_VEL
LIN {X 0,Y 658.316,Z 1076.069,A -85,B 0,C 180,E1 30002.467,E2 30002.467} C_VEL
LIN {X 0,Y 656.556,Z 1097.844,A -85,B 0,C 180,E1 30000.771,E2 30000.771} C_VEL
LIN {X 0,Y 654.872,Z 1118.114,A -85,B 0,C 180,E1 29998.968,E2 29998.968} C_VEL
LIN {X 0,Y 653.547,Z 1134.616,A -85,B 0,C 180,E1 29997.342,E2 29997.342} C_VEL
LIN {X 0,Y 652.208,Z 1153.08,A -85,B 0,C 180,E1 29995.318,E2 29995.318} C_VEL
LIN {X 0,Y 651.017,Z 1169.69,A -85,B 0,C 180,E1 29993.243,E2 29993.243} C_VEL
LIN {X 0,Y 650.201,Z 1183.119,A -85,B 0,C 180,E1 29991.369,E2 29991.369} C_VEL
LIN {X 0,Y 649.418,Z 1197.876,A -85,B 0,C 180,E1 29989.046,E2 29989.046} C_VEL
LIN {X 0,Y 648.827,Z 1209.944,A -85,B 0,C 180,E1 29986.836,E2 29986.836} C_VEL
LIN {X 0,Y 648.508,Z 1219.127,A -85,B 0,C 180,E1 29984.916,E2 29984.916} C_VEL
LIN {X 0,Y 648.252,Z 1227.773,A -85,B 0,C 180,E1 29982.828,E2 29982.828} C_VEL
LIN {X 0,Y 648.06,Z 1236.402,A -85,B 0,C 180,E1 29980.305,E2 29980.305} C_VEL
LIN {X 0,Y 647.947,Z 1242.442,A -85,B 0,C 180,E1 29978.068,E2 29978.068} C_VEL
LIN {X 0,Y 647.929,Z 1246.972,A -85,B 0,C 180,E1 29975.841,E2 29975.841} C_VEL
LIN {X 0,Y 647.912,Z 1250.237,A -85,B 0,C 180,E1 29973.446,E2 29973.446} C_VEL
LIN {X 0,Y 647.889,Z 1251.704,A -85,B 0,C 180,E1 29971.145,E2 29971.145} C_VEL
LIN {X 0,Y 647.864,Z 1251.837,A -85,B 0,C 180,E1 29969.289,E2 29969.289} C_VEL
LIN {X 0,Y 647.904,Z 1250.978,A -85,B 0,C 180,E1 29967.431,E2 29967.431} C_VEL
LIN {X 0,Y 647.911,Z 1248.961,A -85,B 0,C 180,E1 29965.393,E2 29965.393} C_VEL
LIN {X 0,Y 647.935,Z 1245.158,A -85,B 0,C 180,E1 29963.083,E2 29963.083} C_VEL
LIN {X 0,Y 647.956,Z 1239.956,A -85,B 0,C 180,E1 29960.851,E2 29960.851} C_VEL
LIN {X 0,Y 648.093,Z 1233.498,A -85,B 0,C 180,E1 29958.697,E2 29958.697} C_VEL
LIN {X 0,Y 648.265,Z 1226.364,A -85,B 0,C 180,E1 29956.721,E2 29956.721} C_VEL
LIN {X 0,Y 648.52,Z 1218.261,A -85,B 0,C 180,E1 29954.802,E2 29954.802} C_VEL
LIN {X 0,Y 648.941,Z 1208.026,A -85,B 0,C 180,E1 29952.697,E2 29952.697} C_VEL
LIN {X 0,Y 649.586,Z 1194.416,A -85,B 0,C 180,E1 29950.297,E2 29950.297} C_VEL
LIN {X 0,Y 650.286,Z 1181.75,A -85,B 0,C 180,E1 29948.341,E2 29948.341} C_VEL
LIN {X 0,Y 651.181,Z 1167.45,A -85,B 0,C 180,E1 29946.371,E2 29946.371} C_VEL
LIN {X 0,Y 652.407,Z 1149.59,A -85,B 0,C 180,E1 29944.195,E2 29944.195} C_VEL
LIN {X 0,Y 653.642,Z 1133.493,A -85,B 0,C 180,E1 29942.452,E2 29942.452} C_VEL
LIN {X 0,Y 654.969,Z 1116.997,A -85,B 0,C 180,E1 29940.836,E2 29940.836} C_VEL
LIN {X 0,Y 656.744,Z 1095.182,A -85,B 0,C 180,E1 29938.925,E2 29938.925} C_VEL
LIN {X 0,Y 658.402,Z 1075.115,A -85,B 0,C 180,E1 29937.373,E2 29937.373} C_VEL
LIN {X 0,Y 660.069,Z 1055.45,A -85,B 0,C 180,E1 29936.013,E2 29936.013} C_VEL
LIN {X 0,Y 662.111,Z 1030.708,A -85,B 0,C 180,E1 29934.501,E2 29934.501} C_VEL
LIN {X 0,Y 663.87,Z 1007.487,A -85,B 0,C 180,E1 29933.275,E2 29933.275} C_VEL
LIN {X 0,Y 665.409,Z 986.209,A -85,B 0,C 180,E1 29932.293,E2 29932.293} C_VEL
LIN {X 0,Y 667.078,Z 961.574,A -85,B 0,C 180,E1 29931.312,E2 29931.312} C_VEL
LIN {X 0,Y 668.667,Z 934.267,A -85,B 0,C 180,E1 29930.424,E2 29930.424} C_VEL
LIN {X 0,Y 669.806,Z 910.95,A -85,B 0,C 180,E1 29929.812,E2 29929.812} C_VEL
LIN {X 0,Y 670.838,Z 885.596,A -85,B 0,C 180,E1 29929.291,E2 29929.291} C_VEL
LIN {X 0,Y 671.666,Z 850.719,A -85,B 0,C 180,E1 29928.792,E2 29928.792} C_VEL
LIN {X 0,Y 675.025,Z 627.761,A -85,B 0,C 180,E1 29925.89,E2 29925.89} C_VEL
LIN {X 0,Y 677.99,Z 442.146,A -85,B 0,C 180,E1 29923.399,E2 29923.399} C_VEL
LIN {X 0,Y 667.44,Z 426.521,A -85,B 0,C 180,E1 29922.185,E2 29922.185} C_VEL
LIN {X 0,Y 659.611,Z 416.092,A -85,B 0,C 180,E1 29921.255,E2 29921.255} C_VEL
LIN {X 0,Y 656.125,Z 411.356,A -85,B 0,C 180,E1 29920.827,E2 29920.827} C_VEL
LIN {X 0,Y 653.257,Z 407.607,A -85,B 0,C 180,E1 29920.47,E2 29920.47} C_VEL
LIN {X 0,Y 652.244,Z 406.067,A -85,B 0,C 180,E1 29920.339,E2 29920.339} C_VEL
LIN {X 0,Y 649.76,Z 403.423,A -85,B 0,C 180,E1 29920.034,E2 29920.034} C_VEL
LIN {X 0,Y 648.751,Z 400.421,A -85,B 0,C 180,E1 29919.864,E2 29919.864} C_VEL
LIN {X 0,Y 648.752,Z 400.421,A -85,B 0,C 180,E1 29916.838,E2 29916.838} C_VEL
LIN {X 0,Y 648.752,Z 400.4,A -85,B 0,C 180,E1 29913.807,E2 29913.807} C_VEL
LIN {X 0,Y 648.755,Z 400.393,A -85,B 0,C 180,E1 29910.777,E2 29910.777} C_VEL
LIN {X 0,Y 648.754,Z 400.417,A -85,B 0,C 180,E1 29907.64,E2 29907.64} C_VEL
LIN {X 0,Y 648.759,Z 400.399,A -85,B 0,C 180,E1 29904.585,E2 29904.585} C_VEL
LIN {X 0,Y 648.758,Z 400.407,A -85,B 0,C 180,E1 29901.519,E2 29901.519} C_VEL
LIN {X 0,Y 648.765,Z 400.413,A -85,B 0,C 180,E1 29898.418,E2 29898.418} C_VEL
LIN {X 0,Y 648.749,Z 400.393,A -85,B 0,C 180,E1 29895.238,E2 29895.238} C_VEL
LIN {X 0,Y 648.767,Z 400.42,A -85,B 0,C 180,E1 29892.19,E2 29892.19} C_VEL
LIN {X 0,Y 648.748,Z 400.386,A -85,B 0,C 180,E1 29889.045,E2 29889.045} C_VEL
LIN {X 0,Y 648.768,Z 400.421,A -85,B 0,C 180,E1 29886.016,E2 29886.016} C_VEL
LIN {X 0,Y 648.745,Z 400.384,A -85,B 0,C 180,E1 29882.827,E2 29882.827} C_VEL
LIN {X 0,Y 648.77,Z 400.42,A -85,B 0,C 180,E1 29879.735,E2 29879.735} C_VEL
LIN {X 0,Y 648.741,Z 400.382,A -85,B 0,C 180,E1 29876.554,E2 29876.554} C_VEL
LIN {X 0,Y 648.768,Z 400.417,A -85,B 0,C 180,E1 29873.451,E2 29873.451} C_VEL
LIN {X 0,Y 648.739,Z 400.388,A -85,B 0,C 180,E1 29870.328,E2 29870.328} C_VEL
LIN {X 0,Y 648.767,Z 400.414,A -85,B 0,C 180,E1 29867.268,E2 29867.268} C_VEL
LIN {X 0,Y 648.74,Z 400.401,A -85,B 0,C 180,E1 29864.106,E2 29864.106} C_VEL
LIN {X 0,Y 648.763,Z 400.404,A -85,B 0,C 180,E1 29861.116,E2 29861.116} C_VEL
LIN {X 0,Y 648.746,Z 400.414,A -85,B 0,C 180,E1 29858.005,E2 29858.005} C_VEL
LIN {X 0,Y 648.759,Z 400.393,A -85,B 0,C 180,E1 29854.923,E2 29854.923} C_VEL
LIN {X 0,Y 648.742,Z 400.415,A -85,B 0,C 180,E1 29851.76,E2 29851.76} C_VEL
LIN {X 0,Y 648.763,Z 400.412,A -85,B 0,C 180,E1 29848.708,E2 29848.708} C_VEL
LIN {X 0,Y 648.739,Z 400.399,A -85,B 0,C 180,E1 29845.549,E2 29845.549} C_VEL
LIN {X 0,Y 648.753,Z 400.393,A -85,B 0,C 180,E1 29842.539,E2 29842.539} C_VEL
LIN {X 0,Y 648.791,Z 400.569,A -85,B 0,C 180,E1 29842.327,E2 29842.327} C_VEL
LIN {X 0,Y 650,Z 403.769,A -85,B 0,C 180,E1 29841.913,E2 29841.913} C_VEL
LIN {X 0,Y 651.038,Z 405.517,A -85,B 0,C 180,E1 29841.649,E2 29841.649} C_VEL
LIN {X 0,Y 657.863,Z 419.841,A -85,B 0,C 180,E1 29839.731,E2 29839.731} C_VEL
LIN {X 0,Y 661.685,Z 427.475,A -85,B 0,C 180,E1 29838.773,E2 29838.773} C_VEL
LIN {X 0,Y 675.93,Z 448.267,A -85,B 0,C 180,E1 29837.105,E2 29837.105} C_VEL
LIN {X 0,Y 678.28,Z 458.646,A -85,B 0,C 180,E1 29836.734,E2 29836.734} C_VEL
LIN {X 0,Y 674.873,Z 667.235,A -85,B 0,C 180,E1 29833.941,E2 29833.941} C_VEL
LIN {X 0,Y 671.489,Z 892.594,A -85,B 0,C 180,E1 29831.01,E2 29831.01} C_VEL
LIN {X 0,Y 670.673,Z 919.853,A -85,B 0,C 180,E1 29830.584,E2 29830.584} C_VEL
LIN {X 0,Y 669.706,Z 943.182,A -85,B 0,C 180,E1 29830.09,E2 29830.09} C_VEL
LIN {X 0,Y 668.43,Z 968.985,A -85,B 0,C 180,E1 29829.395,E2 29829.395} C_VEL
LIN {X 0,Y 666.805,Z 995.667,A -85,B 0,C 180,E1 29828.486,E2 29828.486} C_VEL
LIN {X 0,Y 665.325,Z 1017.534,A -85,B 0,C 180,E1 29827.603,E2 29827.603} C_VEL
LIN {X 0,Y 663.793,Z 1038.655,A -85,B 0,C 180,E1 29826.622,E2 29826.622} C_VEL
LIN {X 0,Y 661.91,Z 1063.473,A -85,B 0,C 180,E1 29825.299,E2 29825.299} C_VEL
LIN {X 0,Y 659.976,Z 1086.457,A -85,B 0,C 180,E1 29823.876,E2 29823.876} C_VEL
LIN {X 0,Y 658.336,Z 1105.867,A -85,B 0,C 180,E1 29822.527,E2 29822.527} C_VEL
LIN {X 0,Y 656.539,Z 1128.036,A -85,B 0,C 180,E1 29820.8,E2 29820.8} C_VEL
LIN {X 0,Y 654.905,Z 1147.736,A -85,B 0,C 180,E1 29819.049,E2 29819.049} C_VEL
LIN {X 0,Y 653.574,Z 1164.28,A -85,B 0,C 180,E1 29817.422,E2 29817.422} C_VEL
LIN {X 0,Y 652.24,Z 1182.579,A -85,B 0,C 180,E1 29815.422,E2 29815.422} C_VEL
LIN {X 0,Y 651.022,Z 1199.612,A -85,B 0,C 180,E1 29813.298,E2 29813.298} C_VEL
LIN {X 0,Y 650.226,Z 1212.726,A -85,B 0,C 180,E1 29811.471,E2 29811.471} C_VEL
LIN {X 0,Y 649.468,Z 1227.006,A -85,B 0,C 180,E1 29809.239,E2 29809.239} C_VEL
LIN {X 0,Y 648.846,Z 1239.661,A -85,B 0,C 180,E1 29806.936,E2 29806.936} C_VEL
LIN {X 0,Y 648.512,Z 1248.881,A -85,B 0,C 180,E1 29805.016,E2 29805.016} C_VEL
LIN {X 0,Y 648.26,Z 1257.211,A -85,B 0,C 180,E1 29803.018,E2 29803.018} C_VEL
LIN {X 0,Y 648.065,Z 1265.588,A -85,B 0,C 180,E1 29800.635,E2 29800.635} C_VEL
LIN {X 0,Y 647.958,Z 1272.321,A -85,B 0,C 180,E1 29798.165,E2 29798.165} C_VEL
LIN {X 0,Y 647.93,Z 1276.879,A -85,B 0,C 180,E1 29795.938,E2 29795.938} C_VEL
LIN {X 0,Y 647.914,Z 1280.19,A -85,B 0,C 180,E1 29793.543,E2 29793.543} C_VEL
LIN {X 0,Y 647.893,Z 1281.691,A -85,B 0,C 180,E1 29791.242,E2 29791.242} C_VEL
LIN {X 0,Y 647.864,Z 1281.85,A -85,B 0,C 180,E1 29789.385,E2 29789.385} C_VEL
LIN {X 0,Y 647.906,Z 1281.017,A -85,B 0,C 180,E1 29787.528,E2 29787.528} C_VEL
LIN {X 0,Y 647.913,Z 1279.026,A -85,B 0,C 180,E1 29785.49,E2 29785.49} C_VEL
LIN {X 0,Y 647.936,Z 1275.259,A -85,B 0,C 180,E1 29783.18,E2 29783.18} C_VEL
LIN {X 0,Y 647.955,Z 1269.851,A -85,B 0,C 180,E1 29780.859,E2 29780.859} C_VEL
LIN {X 0,Y 648.1,Z 1263.373,A -85,B 0,C 180,E1 29778.705,E2 29778.705} C_VEL
LIN {X 0,Y 648.264,Z 1256.531,A -85,B 0,C 180,E1 29776.809,E2 29776.809} C_VEL
LIN {X 0,Y 648.528,Z 1248.098,A -85,B 0,C 180,E1 29774.81,E2 29774.81} C_VEL
LIN {X 0,Y 648.97,Z 1237.379,A -85,B 0,C 180,E1 29772.614,E2 29772.614} C_VEL
LIN {X 0,Y 649.598,Z 1224.195,A -85,B 0,C 180,E1 29770.306,E2 29770.306} C_VEL
LIN {X 0,Y 650.3,Z 1211.504,A -85,B 0,C 180,E1 29768.35,E2 29768.35} C_VEL
LIN {X 0,Y 651.201,Z 1197.181,A -85,B 0,C 180,E1 29766.381,E2 29766.381} C_VEL
LIN {X 0,Y 652.426,Z 1179.277,A -85,B 0,C 180,E1 29764.205,E2 29764.205} C_VEL
LIN {X 0,Y 653.685,Z 1162.992,A -85,B 0,C 180,E1 29762.446,E2 29762.446} C_VEL
LIN {X 0,Y 655.116,Z 1145.29,A -85,B 0,C 180,E1 29760.72,E2 29760.72} C_VEL
LIN {X 0,Y 656.894,Z 1123.187,A -85,B 0,C 180,E1 29758.81,E2 29758.81} C_VEL
LIN {X 0,Y 658.442,Z 1104.651,A -85,B 0,C 180,E1 29757.385,E2 29757.385} C_VEL
LIN {X 0,Y 660.113,Z 1084.946,A -85,B 0,C 180,E1 29756.025,E2 29756.025} C_VEL
LIN {X 0,Y 662.149,Z 1060.115,A -85,B 0,C 180,E1 29754.513,E2 29754.513} C_VEL
LIN {X 0,Y 663.848,Z 1037.838,A -85,B 0,C 180,E1 29753.337,E2 29753.337} C_VEL
LIN {X 0,Y 665.411,Z 1016.2,A -85,B 0,C 180,E1 29752.338,E2 29752.338} C_VEL
LIN {X 0,Y 667.106,Z 991.205,A -85,B 0,C 180,E1 29751.343,E2 29751.343} C_VEL
LIN {X 0,Y 668.679,Z 963.988,A -85,B 0,C 180,E1 29750.461,E2 29750.461} C_VEL
LIN {X 0,Y 669.817,Z 940.7,A -85,B 0,C 180,E1 29749.851,E2 29749.851} C_VEL
LIN {X 0,Y 670.865,Z 915.03,A -85,B 0,C 180,E1 29749.326,E2 29749.326} C_VEL
LIN {X 0,Y 671.684,Z 879.501,A -85,B 0,C 180,E1 29748.822,E2 29748.822} C_VEL
LIN {X 0,Y 675.072,Z 654.877,A -85,B 0,C 180,E1 29745.897,E2 29745.897} C_VEL
LIN {X 0,Y 678.256,Z 457.737,A -85,B 0,C 180,E1 29743.25,E2 29743.25} C_VEL
LIN {X 0,Y 675.636,Z 447.755,A -85,B 0,C 180,E1 29742.86,E2 29742.86} C_VEL
LIN {X 0,Y 661.187,Z 426.486,A -85,B 0,C 180,E1 29741.135,E2 29741.135} C_VEL
LIN {X 0,Y 654.17,Z 412.219,A -85,B 0,C 180,E1 29739.257,E2 29739.257} C_VEL
LIN {X 0,Y 652.229,Z 408.283,A -85,B 0,C 180,E1 29738.718,E2 29738.718} C_VEL
LIN {X 0,Y 650.373,Z 404.292,A -85,B 0,C 180,E1 29738.173,E2 29738.173} C_VEL
LIN {X 0,Y 648.853,Z 401.002,A -85,B 0,C 180,E1 29737.719,E2 29737.719} C_VEL
LIN {X 0,Y 648.74,Z 400.395,A -85,B 0,C 180,E1 29737.615,E2 29737.615} C_VEL
LIN {X 0,Y 648.707,Z 400.409,A -85,B 0,C 180,E1 29734.772,E2 29734.772} C_VEL
LIN {X 0,Y 648.767,Z 400.42,A -85,B 0,C 180,E1 29731.706,E2 29731.706} C_VEL
LIN {X 0,Y 648.695,Z 400.411,A -85,B 0,C 180,E1 29728.846,E2 29728.846} C_VEL
LIN {X 0,Y 648.738,Z 400.402,A -85,B 0,C 180,E1 29726.046,E2 29726.046} C_VEL
LIN {X 0,Y 648.696,Z 400.425,A -85,B 0,C 180,E1 29722.953,E2 29722.953} C_VEL
LIN {X 0,Y 648.684,Z 400.397,A -85,B 0,C 180,E1 29720.387,E2 29720.387} C_VEL
LIN {X 0,Y 648.755,Z 400.422,A -85,B 0,C 180,E1 29717.398,E2 29717.398} C_VEL
LIN {X 0,Y 648.671,Z 400.4,A -85,B 0,C 180,E1 29714.552,E2 29714.552} C_VEL
LIN {X 0,Y 648.688,Z 400.425,A -85,B 0,C 180,E1 29711.92,E2 29711.92} C_VEL
LIN {X 0,Y 648.676,Z 400.401,A -85,B 0,C 180,E1 29708.688,E2 29708.688} C_VEL
LIN {X 0,Y 648.662,Z 400.426,A -85,B 0,C 180,E1 29706.194,E2 29706.194} C_VEL
LIN {X 0,Y 648.726,Z 400.394,A -85,B 0,C 180,E1 29703.358,E2 29703.358} C_VEL
LIN {X 0,Y 648.681,Z 400.425,A -85,B 0,C 180,E1 29700.353,E2 29700.353} C_VEL
LIN {X 0,Y 648.678,Z 400.406,A -85,B 0,C 180,E1 29697.791,E2 29697.791} C_VEL
LIN {X 0,Y 648.755,Z 400.418,A -85,B 0,C 180,E1 29694.783,E2 29694.783} C_VEL
LIN {X 0,Y 648.685,Z 400.409,A -85,B 0,C 180,E1 29691.937,E2 29691.937} C_VEL
LIN {X 0,Y 648.728,Z 400.411,A -85,B 0,C 180,E1 29689.162,E2 29689.162} C_VEL
LIN {X 0,Y 648.708,Z 400.404,A -85,B 0,C 180,E1 29686.087,E2 29686.087} C_VEL
LIN {X 0,Y 648.702,Z 400.413,A -85,B 0,C 180,E1 29683.432,E2 29683.432} C_VEL
LIN {X 0,Y 648.764,Z 400.392,A -85,B 0,C 180,E1 29680.367,E2 29680.367} C_VEL
LIN {X 0,Y 648.709,Z 400.419,A -85,B 0,C 180,E1 29677.39,E2 29677.39} C_VEL
LIN {X 0,Y 648.77,Z 400.39,A -85,B 0,C 180,E1 29674.354,E2 29674.354} C_VEL
LIN {X 0,Y 648.718,Z 400.421,A -85,B 0,C 180,E1 29671.357,E2 29671.357} C_VEL
LIN {X 0,Y 648.769,Z 400.404,A -85,B 0,C 180,E1 29668.398,E2 29668.398} C_VEL
LIN {X 0,Y 648.725,Z 400.394,A -85,B 0,C 180,E1 29665.337,E2 29665.337} C_VEL
LIN {X 0,Y 648.767,Z 400.399,A -85,B 0,C 180,E1 29662.379,E2 29662.379} C_VEL
LIN {X 0,Y 648.793,Z 400.617,A -85,B 0,C 180,E1 29660.026,E2 29660.026} C_VEL
LIN {X 0,Y 649.953,Z 403.72,A -85,B 0,C 180,E1 29659.85,E2 29659.85} C_VEL
LIN {X 0,Y 652.944,Z 406.999,A -85,B 0,C 180,E1 29659.482,E2 29659.482} C_VEL
LIN {X 0,Y 655.657,Z 410.928,A -85,B 0,C 180,E1 29659.138,E2 29659.138} C_VEL
LIN {X 0,Y 657.272,Z 412.84,A -85,B 0,C 180,E1 29658.943,E2 29658.943} C_VEL
LIN {X 0,Y 664.204,Z 422.006,A -85,B 0,C 180,E1 29658.108,E2 29658.108} C_VEL
LIN {X 0,Y 665.975,Z 425.145,A -85,B 0,C 180,E1 29657.887,E2 29657.887} C_VEL
LIN {X 0,Y 667.436,Z 431.993,A -85,B 0,C 180,E1 29657.639,E2 29657.639} C_VEL
LIN {X 0,Y 668.913,Z 439.789,A -85,B 0,C 180,E1 29657.378,E2 29657.378} C_VEL
LIN {X 0,Y 670.262,Z 442.716,A -85,B 0,C 180,E1 29657.206,E2 29657.206} C_VEL
LIN {X 0,Y 672.466,Z 446.298,A -85,B 0,C 180,E1 29656.947,E2 29656.947} C_VEL
LIN {X 0,Y 668.835,Z 653.547,A -85,B 0,C 180,E1 29654.156,E2 29654.156} C_VEL
LIN {X 0,Y 665.203,Z 871.194,A -85,B 0,C 180,E1 29651.297,E2 29651.297} C_VEL
LIN {X 0,Y 664.383,Z 894.578,A -85,B 0,C 180,E1 29650.901,E2 29650.901} C_VEL
LIN {X 0,Y 663.154,Z 921.695,A -85,B 0,C 180,E1 29650.286,E2 29650.286} C_VEL
LIN {X 0,Y 661.643,Z 947.085,A -85,B 0,C 180,E1 29649.534,E2 29649.534} C_VEL
LIN {X 0,Y 660.305,Z 967.423,A -85,B 0,C 180,E1 29648.815,E2 29648.815} C_VEL
LIN {X 0,Y 658.803,Z 987.949,A -85,B 0,C 180,E1 29647.976,E2 29647.976} C_VEL
LIN {X 0,Y 657.084,Z 1010.012,A -85,B 0,C 180,E1 29646.939,E2 29646.939} C_VEL
LIN {X 0,Y 654.938,Z 1035.717,A -85,B 0,C 180,E1 29645.538,E2 29645.538} C_VEL
LIN {X 0,Y 653.072,Z 1056.549,A -85,B 0,C 180,E1 29644.231,E2 29644.231} C_VEL
LIN {X 0,Y 651.323,Z 1075.723,A -85,B 0,C 180,E1 29642.887,E2 29642.887} C_VEL
LIN {X 0,Y 649.403,Z 1097.253,A -85,B 0,C 180,E1 29641.199,E2 29641.199} C_VEL
LIN {X 0,Y 647.559,Z 1117.887,A -85,B 0,C 180,E1 29639.35,E2 29639.35} C_VEL
LIN {X 0,Y 646.147,Z 1134.181,A -85,B 0,C 180,E1 29637.729,E2 29637.729} C_VEL
LIN {X 0,Y 644.644,Z 1152.679,A -85,B 0,C 180,E1 29635.687,E2 29635.687} C_VEL
LIN {X 0,Y 643.338,Z 1169.696,A -85,B 0,C 180,E1 29633.537,E2 29633.537} C_VEL
LIN {X 0,Y 642.438,Z 1183.121,A -85,B 0,C 180,E1 29631.64,E2 29631.64} C_VEL
LIN {X 0,Y 641.576,Z 1197.881,A -85,B 0,C 180,E1 29629.288,E2 29629.288} C_VEL
LIN {X 0,Y 640.936,Z 1209.949,A -85,B 0,C 180,E1 29627.05,E2 29627.05} C_VEL
LIN {X 0,Y 640.563,Z 1219.131,A -85,B 0,C 180,E1 29625.105,E2 29625.105} C_VEL
LIN {X 0,Y 640.286,Z 1227.421,A -85,B 0,C 180,E1 29623.082,E2 29623.082} C_VEL
LIN {X 0,Y 640.078,Z 1235.892,A -85,B 0,C 180,E1 29620.617,E2 29620.617} C_VEL
LIN {X 0,Y 639.959,Z 1242.441,A -85,B 0,C 180,E1 29618.169,E2 29618.169} C_VEL
LIN {X 0,Y 639.931,Z 1246.97,A -85,B 0,C 180,E1 29615.915,E2 29615.915} C_VEL
LIN {X 0,Y 639.912,Z 1250.237,A -85,B 0,C 180,E1 29613.489,E2 29613.489} C_VEL
LIN {X 0,Y 639.89,Z 1251.704,A -85,B 0,C 180,E1 29611.16,E2 29611.16} C_VEL
LIN {X 0,Y 639.864,Z 1251.837,A -85,B 0,C 180,E1 29609.28,E2 29609.28} C_VEL
LIN {X 0,Y 639.905,Z 1250.978,A -85,B 0,C 180,E1 29607.399,E2 29607.399} C_VEL
LIN {X 0,Y 639.911,Z 1248.957,A -85,B 0,C 180,E1 29605.336,E2 29605.336} C_VEL
LIN {X 0,Y 639.939,Z 1245.157,A -85,B 0,C 180,E1 29602.996,E2 29602.996} C_VEL
LIN {X 0,Y 639.962,Z 1239.954,A -85,B 0,C 180,E1 29600.736,E2 29600.736} C_VEL
LIN {X 0,Y 640.121,Z 1233.495,A -85,B 0,C 180,E1 29598.554,E2 29598.554} C_VEL
LIN {X 0,Y 640.291,Z 1226.658,A -85,B 0,C 180,E1 29596.629,E2 29596.629} C_VEL
LIN {X 0,Y 640.568,Z 1218.671,A -85,B 0,C 180,E1 29594.701,E2 29594.701} C_VEL
LIN {X 0,Y 641.001,Z 1208.955,A -85,B 0,C 180,E1 29592.663,E2 29592.663} C_VEL
LIN {X 0,Y 641.698,Z 1195.557,A -85,B 0,C 180,E1 29590.234,E2 29590.234} C_VEL
LIN {X 0,Y 642.49,Z 1182.387,A -85,B 0,C 180,E1 29588.161,E2 29588.161} C_VEL
LIN {X 0,Y 643.408,Z 1168.809,A -85,B 0,C 180,E1 29586.254,E2 29586.254} C_VEL
LIN {X 0,Y 644.73,Z 1151.274,A -85,B 0,C 180,E1 29584.063,E2 29584.063} C_VEL
LIN {X 0,Y 646.186,Z 1133.768,A -85,B 0,C 180,E1 29582.138,E2 29582.138} C_VEL
LIN {X 0,Y 647.624,Z 1117.17,A -85,B 0,C 180,E1 29580.491,E2 29580.491} C_VEL
LIN {X 0,Y 649.517,Z 1095.78,A -85,B 0,C 180,E1 29578.591,E2 29578.591} C_VEL
LIN {X 0,Y 651.32,Z 1075.772,A -85,B 0,C 180,E1 29577.026,E2 29577.026} C_VEL
LIN {X 0,Y 653.039,Z 1056.907,A -85,B 0,C 180,E1 29575.702,E2 29575.702} C_VEL
LIN {X 0,Y 655.058,Z 1034.478,A -85,B 0,C 180,E1 29574.297,E2 29574.297} C_VEL
LIN {X 0,Y 657.122,Z 1009.478,A -85,B 0,C 180,E1 29572.944,E2 29572.944} C_VEL
LIN {X 0,Y 658.766,Z 988.452,A -85,B 0,C 180,E1 29571.956,E2 29571.956} C_VEL
LIN {X 0,Y 660.348,Z 966.694,A -85,B 0,C 180,E1 29571.066,E2 29571.066} C_VEL
LIN {X 0,Y 662.052,Z 941.112,A -85,B 0,C 180,E1 29570.179,E2 29570.179} C_VEL
LIN {X 0,Y 663.498,Z 914.156,A -85,B 0,C 180,E1 29569.439,E2 29569.439} C_VEL
LIN {X 0,Y 664.536,Z 890.762,A -85,B 0,C 180,E1 29568.937,E2 29568.937} C_VEL
LIN {X 0,Y 665.379,Z 865.339,A -85,B 0,C 180,E1 29568.529,E2 29568.529} C_VEL
LIN {X 0,Y 669.039,Z 641.319,A -85,B 0,C 180,E1 29565.591,E2 29565.591} C_VEL
LIN {X 0,Y 672.466,Z 446.02,A -85,B 0,C 180,E1 29562.959,E2 29562.959} C_VEL
LIN {X 0,Y 662.792,Z 431.798,A -85,B 0,C 180,E1 29561.821,E2 29561.821} C_VEL
LIN {X 0,Y 655.319,Z 421.793,A -85,B 0,C 180,E1 29560.916,E2 29560.916} C_VEL
LIN {X 0,Y 651.85,Z 417.193,A -85,B 0,C 180,E1 29560.484,E2 29560.484} C_VEL
LIN {X 0,Y 648.277,Z 412.383,A -85,B 0,C 180,E1 29560.029,E2 29560.029} C_VEL
LIN {X 0,Y 645.434,Z 408.7,A -85,B 0,C 180,E1 29559.662,E2 29559.662} C_VEL
LIN {X 0,Y 644.617,Z 407.262,A -85,B 0,C 180,E1 29559.55,E2 29559.55} C_VEL
LIN {X 0,Y 641.947,Z 404.6,A -85,B 0,C 180,E1 29559.212,E2 29559.212} C_VEL
LIN {X 0,Y 640.816,Z 401.405,A -85,B 0,C 180,E1 29559.007,E2 29559.007} C_VEL
LIN {X 0,Y 640.817,Z 401.401,A -85,B 0,C 180,E1 29555.92,E2 29555.92} C_VEL
LIN {X 0,Y 640.817,Z 401.409,A -85,B 0,C 180,E1 29552.782,E2 29552.782} C_VEL
LIN {X 0,Y 640.815,Z 401.381,A -85,B 0,C 180,E1 29549.748,E2 29549.748} C_VEL
LIN {X 0,Y 640.823,Z 401.389,A -85,B 0,C 180,E1 29546.704,E2 29546.704} C_VEL
LIN {X 0,Y 640.815,Z 401.402,A -85,B 0,C 180,E1 29543.544,E2 29543.544} C_VEL
LIN {X 0,Y 640.822,Z 401.377,A -85,B 0,C 180,E1 29540.458,E2 29540.458} C_VEL
LIN {X 0,Y 640.812,Z 401.405,A -85,B 0,C 180,E1 29537.264,E2 29537.264} C_VEL
LIN {X 0,Y 640.823,Z 401.379,A -85,B 0,C 180,E1 29534.18,E2 29534.18} C_VEL
LIN {X 0,Y 640.81,Z 401.404,A -85,B 0,C 180,E1 29531.046,E2 29531.046} C_VEL
LIN {X 0,Y 640.823,Z 401.38,A -85,B 0,C 180,E1 29527.982,E2 29527.982} C_VEL
LIN {X 0,Y 640.808,Z 401.403,A -85,B 0,C 180,E1 29524.833,E2 29524.833} C_VEL
LIN {X 0,Y 640.822,Z 401.382,A -85,B 0,C 180,E1 29521.699,E2 29521.699} C_VEL
LIN {X 0,Y 640.808,Z 401.401,A -85,B 0,C 180,E1 29518.659,E2 29518.659} C_VEL
LIN {X 0,Y 640.823,Z 401.382,A -85,B 0,C 180,E1 29515.525,E2 29515.525} C_VEL
LIN {X 0,Y 640.803,Z 401.399,A -85,B 0,C 180,E1 29512.378,E2 29512.378} C_VEL
LIN {X 0,Y 640.825,Z 401.389,A -85,B 0,C 180,E1 29509.299,E2 29509.299} C_VEL
LIN {X 0,Y 640.802,Z 401.395,A -85,B 0,C 180,E1 29506.188,E2 29506.188} C_VEL
LIN {X 0,Y 640.826,Z 401.401,A -85,B 0,C 180,E1 29503.129,E2 29503.129} C_VEL
LIN {X 0,Y 640.797,Z 401.379,A -85,B 0,C 180,E1 29499.946,E2 29499.946} C_VEL
LIN {X 0,Y 640.832,Z 401.407,A -85,B 0,C 180,E1 29496.944,E2 29496.944} C_VEL
LIN {X 0,Y 640.8,Z 401.393,A -85,B 0,C 180,E1 29493.795,E2 29493.795} C_VEL
LIN {X 0,Y 640.822,Z 401.382,A -85,B 0,C 180,E1 29490.766,E2 29490.766} C_VEL
LIN {X 0,Y 640.801,Z 401.407,A -85,B 0,C 180,E1 29487.585,E2 29487.585} C_VEL
LIN {X 0,Y 640.825,Z 401.406,A -85,B 0,C 180,E1 29484.518,E2 29484.518} C_VEL
LIN {X 0,Y 640.8,Z 401.512,A -85,B 0,C 180,E1 29483.138,E2 29483.138} C_VEL
LIN {X 0,Y 642.005,Z 404.714,A -85,B 0,C 180,E1 29482.71,E2 29482.71} C_VEL
LIN {X 0,Y 643.09,Z 406.284,A -85,B 0,C 180,E1 29482.447,E2 29482.447} C_VEL
LIN {X 0,Y 651.344,Z 423.41,A -85,B 0,C 180,E1 29480.083,E2 29480.083} C_VEL
LIN {X 0,Y 653.261,Z 427.172,A -85,B 0,C 180,E1 29479.621,E2 29479.621} C_VEL
LIN {X 0,Y 671.003,Z 452.966,A -85,B 0,C 180,E1 29477.485,E2 29477.485} C_VEL
LIN {X 0,Y 672.752,Z 460.804,A -85,B 0,C 180,E1 29477.204,E2 29477.204} C_VEL
LIN {X 0,Y 669.077,Z 669.089,A -85,B 0,C 180,E1 29474.393,E2 29474.393} C_VEL
LIN {X 0,Y 665.413,Z 894.151,A -85,B 0,C 180,E1 29471.443,E2 29471.443} C_VEL
LIN {X 0,Y 664.559,Z 920.315,A -85,B 0,C 180,E1 29471.026,E2 29471.026} C_VEL
LIN {X 0,Y 663.533,Z 943.422,A -85,B 0,C 180,E1 29470.533,E2 29470.533} C_VEL
LIN {X 0,Y 662.174,Z 969.089,A -85,B 0,C 180,E1 29469.837,E2 29469.837} C_VEL
LIN {X 0,Y 660.421,Z 995.657,A -85,B 0,C 180,E1 29468.928,E2 29468.928} C_VEL
LIN {X 0,Y 658.815,Z 1017.766,A -85,B 0,C 180,E1 29468.029,E2 29468.029} C_VEL
LIN {X 0,Y 657.18,Z 1038.653,A -85,B 0,C 180,E1 29467.052,E2 29467.052} C_VEL
LIN {X 0,Y 655.15,Z 1063.543,A -85,B 0,C 180,E1 29465.714,E2 29465.714} C_VEL
LIN {X 0,Y 653.098,Z 1086.285,A -85,B 0,C 180,E1 29464.294,E2 29464.294} C_VEL
LIN {X 0,Y 651.375,Z 1105.199,A -85,B 0,C 180,E1 29462.971,E2 29462.971} C_VEL
LIN {X 0,Y 649.561,Z 1125.253,A -85,B 0,C 180,E1 29461.406,E2 29461.406} C_VEL
LIN {X 0,Y 647.665,Z 1146.72,A -85,B 0,C 180,E1 29459.507,E2 29459.507} C_VEL
LIN {X 0,Y 646.222,Z 1163.352,A -85,B 0,C 180,E1 29457.861,E2 29457.861} C_VEL
LIN {X 0,Y 644.818,Z 1180.044,A -85,B 0,C 180,E1 29456.032,E2 29456.032} C_VEL
LIN {X 0,Y 643.429,Z 1198.54,A -85,B 0,C 180,E1 29453.737,E2 29453.737} C_VEL
LIN {X 0,Y 642.51,Z 1212.089,A -85,B 0,C 180,E1 29451.838,E2 29451.838} C_VEL
LIN {X 0,Y 641.687,Z 1225.858,A -85,B 0,C 180,E1 29449.672,E2 29449.672} C_VEL
LIN {X 0,Y 640.985,Z 1239.197,A -85,B 0,C 180,E1 29447.244,E2 29447.244} C_VEL
LIN {X 0,Y 640.575,Z 1248.561,A -85,B 0,C 180,E1 29445.278,E2 29445.278} C_VEL
LIN {X 0,Y 640.292,Z 1256.501,A -85,B 0,C 180,E1 29443.366,E2 29443.366} C_VEL
LIN {X 0,Y 640.128,Z 1263.346,A -85,B 0,C 180,E1 29441.445,E2 29441.445} C_VEL
LIN {X 0,Y 639.963,Z 1269.828,A -85,B 0,C 180,E1 29439.264,E2 29439.264} C_VEL
LIN {X 0,Y 639.939,Z 1275.243,A -85,B 0,C 180,E1 29436.914,E2 29436.914} C_VEL
LIN {X 0,Y 639.912,Z 1279.014,A -85,B 0,C 180,E1 29434.575,E2 29434.575} C_VEL
LIN {X 0,Y 639.906,Z 1281.012,A -85,B 0,C 180,E1 29432.512,E2 29432.512} C_VEL
LIN {X 0,Y 639.866,Z 1281.871,A -85,B 0,C 180,E1 29430.541,E2 29430.541} C_VEL
LIN {X 0,Y 639.91,Z 1281.551,A -85,B 0,C 180,E1 29428.213,E2 29428.213} C_VEL
LIN {X 0,Y 639.919,Z 1279.365,A -85,B 0,C 180,E1 29425.703,E2 29425.703} C_VEL
LIN {X 0,Y 639.939,Z 1275.932,A -85,B 0,C 180,E1 29423.455,E2 29423.455} C_VEL
LIN {X 0,Y 639.967,Z 1270.606,A -85,B 0,C 180,E1 29421.016,E2 29421.016} C_VEL
LIN {X 0,Y 640.118,Z 1263.676,A -85,B 0,C 180,E1 29418.654,E2 29418.654} C_VEL
LIN {X 0,Y 640.291,Z 1256.533,A -85,B 0,C 180,E1 29416.642,E2 29416.642} C_VEL
LIN {X 0,Y 640.577,Z 1248.51,A -85,B 0,C 180,E1 29414.71,E2 29414.71} C_VEL
LIN {X 0,Y 641.009,Z 1238.777,A -85,B 0,C 180,E1 29412.672,E2 29412.672} C_VEL
LIN {X 0,Y 641.712,Z 1225.339,A -85,B 0,C 180,E1 29410.243,E2 29410.243} C_VEL
LIN {X 0,Y 642.507,Z 1212.148,A -85,B 0,C 180,E1 29408.17,E2 29408.17} C_VEL
LIN {X 0,Y 643.438,Z 1198.427,A -85,B 0,C 180,E1 29406.248,E2 29406.248} C_VEL
LIN {X 0,Y 644.812,Z 1180.12,A -85,B 0,C 180,E1 29403.976,E2 29403.976} C_VEL
LIN {X 0,Y 646.214,Z 1163.437,A -85,B 0,C 180,E1 29402.148,E2 29402.148} C_VEL
LIN {X 0,Y 647.656,Z 1146.813,A -85,B 0,C 180,E1 29400.502,E2 29400.502} C_VEL
LIN {X 0,Y 649.603,Z 1124.757,A -85,B 0,C 180,E1 29398.554,E2 29398.554} C_VEL
LIN {X 0,Y 651.362,Z 1105.316,A -85,B 0,C 180,E1 29397.038,E2 29397.038} C_VEL
LIN {X 0,Y 653.084,Z 1086.412,A -85,B 0,C 180,E1 29395.715,E2 29395.715} C_VEL
LIN {X 0,Y 655.218,Z 1062.786,A -85,B 0,C 180,E1 29394.242,E2 29394.242} C_VEL
LIN {X 0,Y 657.168,Z 1038.84,A -85,B 0,C 180,E1 29392.957,E2 29392.957} C_VEL
LIN {X 0,Y 658.816,Z 1017.74,A -85,B 0,C 180,E1 29391.969,E2 29391.969} C_VEL
LIN {X 0,Y 660.403,Z 995.892,A -85,B 0,C 180,E1 29391.08,E2 29391.08} C_VEL
LIN {X 0,Y 662.198,Z 968.671,A -85,B 0,C 180,E1 29390.15,E2 29390.15} C_VEL
LIN {X 0,Y 663.54,Z 943.286,A -85,B 0,C 180,E1 29389.463,E2 29389.463} C_VEL
LIN {X 0,Y 664.566,Z 920.142,A -85,B 0,C 180,E1 29388.97,E2 29388.97} C_VEL
LIN {X 0,Y 665.429,Z 893.506,A -85,B 0,C 180,E1 29388.548,E2 29388.548} C_VEL
LIN {X 0,Y 669.106,Z 667.459,A -85,B 0,C 180,E1 29385.585,E2 29385.585} C_VEL
LIN {X 0,Y 672.763,Z 460.08,A -85,B 0,C 180,E1 29382.786,E2 29382.786} C_VEL
LIN {X 0,Y 670.705,Z 452.513,A -85,B 0,C 180,E1 29382.48,E2 29382.48} C_VEL
LIN {X 0,Y 655.838,Z 431.045,A -85,B 0,C 180,E1 29380.704,E2 29380.704} C_VEL
LIN {X 0,Y 652.627,Z 426.233,A -85,B 0,C 180,E1 29380.282,E2 29380.282} C_VEL
LIN {X 0,Y 646.797,Z 414.122,A -85,B 0,C 180,E1 29378.649,E2 29378.649} C_VEL
LIN {X 0,Y 642.746,Z 405.714,A -85,B 0,C 180,E1 29377.464,E2 29377.464} C_VEL
LIN {X 0,Y 641.085,Z 402.835,A -85,B 0,C 180,E1 29377.016,E2 29377.016} C_VEL
LIN {X 0,Y 640.771,Z 401.392,A -85,B 0,C 180,E1 29376.814,E2 29376.814} C_VEL
LIN {X 0,Y 640.822,Z 401.38,A -85,B 0,C 180,E1 29373.744,E2 29373.744} C_VEL
LIN {X 0,Y 640.76,Z 401.402,A -85,B 0,C 180,E1 29370.89,E2 29370.89} C_VEL
LIN {X 0,Y 640.819,Z 401.402,A -85,B 0,C 180,E1 29367.991,E2 29367.991} C_VEL
LIN {X 0,Y 640.752,Z 401.388,A -85,B 0,C 180,E1 29364.919,E2 29364.919} C_VEL
LIN {X 0,Y 640.761,Z 401.413,A -85,B 0,C 180,E1 29362.284,E2 29362.284} C_VEL
LIN {X 0,Y 640.773,Z 401.394,A -85,B 0,C 180,E1 29359.129,E2 29359.129} C_VEL
LIN {X 0,Y 640.737,Z 401.409,A -85,B 0,C 180,E1 29356.407,E2 29356.407} C_VEL
LIN {X 0,Y 640.819,Z 401.39,A -85,B 0,C 180,E1 29353.444,E2 29353.444} C_VEL
LIN {X 0,Y 640.726,Z 401.403,A -85,B 0,C 180,E1 29350.429,E2 29350.429} C_VEL
LIN {X 0,Y 640.75,Z 401.397,A -85,B 0,C 180,E1 29347.713,E2 29347.713} C_VEL
LIN {X 0,Y 640.741,Z 401.4,A -85,B 0,C 180,E1 29344.565,E2 29344.565} C_VEL
LIN {X 0,Y 640.733,Z 401.398,A -85,B 0,C 180,E1 29341.878,E2 29341.878} C_VEL
LIN {X 0,Y 640.802,Z 401.397,A -85,B 0,C 180,E1 29338.838,E2 29338.838} C_VEL
LIN {X 0,Y 640.739,Z 401.396,A -85,B 0,C 180,E1 29335.973,E2 29335.973} C_VEL
LIN {X 0,Y 640.807,Z 401.405,A -85,B 0,C 180,E1 29333.099,E2 29333.099} C_VEL
LIN {X 0,Y 640.755,Z 401.394,A -85,B 0,C 180,E1 29330.025,E2 29330.025} C_VEL
LIN {X 0,Y 640.774,Z 401.414,A -85,B 0,C 180,E1 29327.29,E2 29327.29} C_VEL
LIN {X 0,Y 640.776,Z 401.394,A -85,B 0,C 180,E1 29324.06,E2 29324.06} C_VEL
LIN {X 0,Y 640.773,Z 401.41,A -85,B 0,C 180,E1 29321.273,E2 29321.273} C_VEL
LIN {X 0,Y 640.805,Z 401.399,A -85,B 0,C 180,E1 29318.104,E2 29318.104} C_VEL
LIN {X 0,Y 640.773,Z 401.394,A -85,B 0,C 180,E1 29315.238,E2 29315.238} C_VEL
LIN {X 0,Y 640.83,Z 401.406,A -85,B 0,C 180,E1 29312.089,E2 29312.089} C_VEL
LIN {X 0,Y 640.78,Z 401.383,A -85,B 0,C 180,E1 29309.105,E2 29309.105} C_VEL
LIN {X 0,Y 640.83,Z 401.382,A -85,B 0,C 180,E1 29306.041,E2 29306.041} C_VEL
LIN {X 0,Y 640.791,Z 401.407,A -85,B 0,C 180,E1 29302.964,E2 29302.964} C_VEL
LIN {X 0,Y 640.826,Z 401.631,A -85,B 0,C 180,E1 29300.874,E2 29300.874} C_VEL
LIN {X 0,Y 641.996,Z 404.707,A -85,B 0,C 180,E1 29300.691,E2 29300.691} C_VEL
LIN {X 0,Y 644.751,Z 407.324,A -85,B 0,C 180,E1 29300.345,E2 29300.345} C_VEL
LIN {X 0,Y 647.368,Z 411.468,A -85,B 0,C 180,E1 29299.993,E2 29299.993} C_VEL
LIN {X 0,Y 649.336,Z 413.715,A -85,B 0,C 180,E1 29299.747,E2 29299.747} C_VEL
LIN {X 0,Y 652.718,Z 418.096,A -85,B 0,C 180,E1 29299.321,E2 29299.321} C_VEL
LIN {X 0,Y 666.406,Z 436.79,A -85,B 0,C 180,E1 29297.662,E2 29297.662} C_VEL
LIN {X 0,Y 670.262,Z 442.716,A -85,B 0,C 180,E1 29297.206,E2 29297.206} C_VEL
LIN {X 0,Y 671.064,Z 445.352,A -85,B 0,C 180,E1 29297.09,E2 29297.09} C_VEL
LIN {X 0,Y 670.759,Z 449.988,A -85,B 0,C 180,E1 29297.047,E2 29297.047} C_VEL
LIN {X 0,Y 666.999,Z 463.163,A -85,B 0,C 180,E1 29297.192,E2 29297.192} C_VEL
LIN {X 0,Y 666.637,Z 466.438,A -85,B 0,C 180,E1 29297.175,E2 29297.175} C_VEL
LIN {X 0,Y 662.411,Z 691.872,A -85,B 0,C 180,E1 29294.129,E2 29294.129} C_VEL
LIN {X 0,Y 659.084,Z 874.83,A -85,B 0,C 180,E1 29291.704,E2 29291.704} C_VEL
LIN {X 0,Y 658.048,Z 901.815,A -85,B 0,C 180,E1 29291.216,E2 29291.216} C_VEL
LIN {X 0,Y 656.587,Z 928.22,A -85,B 0,C 180,E1 29290.56,E2 29290.56} C_VEL
LIN {X 0,Y 655.18,Z 950.132,A -85,B 0,C 180,E1 29289.885,E2 29289.885} C_VEL
LIN {X 0,Y 653.766,Z 970.185,A -85,B 0,C 180,E1 29289.156,E2 29289.156} C_VEL
LIN {X 0,Y 652.024,Z 992.473,A -85,B 0,C 180,E1 29288.219,E2 29288.219} C_VEL
LIN {X 0,Y 649.779,Z 1018.62,A -85,B 0,C 180,E1 29286.927,E2 29286.927} C_VEL
LIN {X 0,Y 647.753,Z 1040.243,A -85,B 0,C 180,E1 29285.689,E2 29285.689} C_VEL
LIN {X 0,Y 645.917,Z 1059.468,A -85,B 0,C 180,E1 29284.451,E2 29284.451} C_VEL
LIN {X 0,Y 643.84,Z 1080.723,A -85,B 0,C 180,E1 29282.919,E2 29282.919} C_VEL
LIN {X 0,Y 641.679,Z 1102.864,A -85,B 0,C 180,E1 29281.095,E2 29281.095} C_VEL
LIN {X 0,Y 640.058,Z 1119.9,A -85,B 0,C 180,E1 29279.525,E2 29279.525} C_VEL
LIN {X 0,Y 638.492,Z 1136.728,A -85,B 0,C 180,E1 29277.812,E2 29277.812} C_VEL
LIN {X 0,Y 636.789,Z 1156.213,A -85,B 0,C 180,E1 29275.576,E2 29275.576} C_VEL
LIN {X 0,Y 635.558,Z 1171.113,A -85,B 0,C 180,E1 29273.646,E2 29273.646} C_VEL
LIN {X 0,Y 634.547,Z 1185.155,A -85,B 0,C 180,E1 29271.612,E2 29271.612} C_VEL
LIN {X 0,Y 633.604,Z 1199.976,A -85,B 0,C 180,E1 29269.157,E2 29269.157} C_VEL
LIN {X 0,Y 632.995,Z 1210.884,A -85,B 0,C 180,E1 29267.081,E2 29267.081} C_VEL
LIN {X 0,Y 632.59,Z 1220.351,A -85,B 0,C 180,E1 29265.019,E2 29265.019} C_VEL
LIN {X 0,Y 632.237,Z 1230.167,A -85,B 0,C 180,E1 29262.508,E2 29262.508} C_VEL
LIN {X 0,Y 632.068,Z 1237.431,A -85,B 0,C 180,E1 29260.201,E2 29260.201} C_VEL
LIN {X 0,Y 631.947,Z 1243.058,A -85,B 0,C 180,E1 29257.999,E2 29257.999} C_VEL
LIN {X 0,Y 631.927,Z 1247.567,A -85,B 0,C 180,E1 29255.625,E2 29255.625} C_VEL
LIN {X 0,Y 631.909,Z 1250.441,A -85,B 0,C 180,E1 29253.261,E2 29253.261} C_VEL
LIN {X 0,Y 631.892,Z 1251.704,A -85,B 0,C 180,E1 29251.174,E2 29251.174} C_VEL
LIN {X 0,Y 631.864,Z 1251.837,A -85,B 0,C 180,E1 29249.271,E2 29249.271} C_VEL
LIN {X 0,Y 631.906,Z 1250.978,A -85,B 0,C 180,E1 29247.366,E2 29247.366} C_VEL
LIN {X 0,Y 631.913,Z 1248.953,A -85,B 0,C 180,E1 29245.276,E2 29245.276} C_VEL
LIN {X 0,Y 631.946,Z 1245.156,A -85,B 0,C 180,E1 29242.907,E2 29242.907} C_VEL
LIN {X 0,Y 631.97,Z 1239.952,A -85,B 0,C 180,E1 29240.617,E2 29240.617} C_VEL
LIN {X 0,Y 632.15,Z 1233.493,A -85,B 0,C 180,E1 29238.408,E2 29238.408} C_VEL
LIN {X 0,Y 632.323,Z 1226.673,A -85,B 0,C 180,E1 29236.462,E2 29236.462} C_VEL
LIN {X 0,Y 632.634,Z 1218.669,A -85,B 0,C 180,E1 29234.504,E2 29234.504} C_VEL
LIN {X 0,Y 633.107,Z 1208.953,A -85,B 0,C 180,E1 29232.44,E2 29232.44} C_VEL
LIN {X 0,Y 633.869,Z 1195.551,A -85,B 0,C 180,E1 29229.98,E2 29229.98} C_VEL
LIN {X 0,Y 634.756,Z 1182.222,A -85,B 0,C 180,E1 29227.857,E2 29227.857} C_VEL
LIN {X 0,Y 635.811,Z 1168.155,A -85,B 0,C 180,E1 29225.862,E2 29225.862} C_VEL
LIN {X 0,Y 637.264,Z 1150.355,A -85,B 0,C 180,E1 29223.628,E2 29223.628} C_VEL
LIN {X 0,Y 638.761,Z 1133.76,A -85,B 0,C 180,E1 29221.785,E2 29221.785} C_VEL
LIN {X 0,Y 640.313,Z 1117.163,A -85,B 0,C 180,E1 29220.12,E2 29220.12} C_VEL
LIN {X 0,Y 642.382,Z 1095.725,A -85,B 0,C 180,E1 29218.198,E2 29218.198} C_VEL
LIN {X 0,Y 644.361,Z 1075.465,A -85,B 0,C 180,E1 29216.6,E2 29216.6} C_VEL
LIN {X 0,Y 646.173,Z 1056.895,A -85,B 0,C 180,E1 29215.286,E2 29215.286} C_VEL
LIN {X 0,Y 648.242,Z 1035.392,A -85,B 0,C 180,E1 29213.926,E2 29213.926} C_VEL
LIN {X 0,Y 650.547,Z 1009.464,A -85,B 0,C 180,E1 29212.506,E2 29212.506} C_VEL
LIN {X 0,Y 652.31,Z 988.434,A -85,B 0,C 180,E1 29211.511,E2 29211.511} C_VEL
LIN {X 0,Y 653.914,Z 967.961,A -85,B 0,C 180,E1 29210.666,E2 29210.666} C_VEL
LIN {X 0,Y 655.503,Z 945.535,A -85,B 0,C 180,E1 29209.871,E2 29209.871} C_VEL
LIN {X 0,Y 657.199,Z 917.768,A -85,B 0,C 180,E1 29209.069,E2 29209.069} C_VEL
LIN {X 0,Y 658.391,Z 892.88,A -85,B 0,C 180,E1 29208.518,E2 29208.518} C_VEL
LIN {X 0,Y 659.227,Z 869.984,A -85,B 0,C 180,E1 29208.135,E2 29208.135} C_VEL
LIN {X 0,Y 663.154,Z 650.359,A -85,B 0,C 180,E1 29205.227,E2 29205.227} C_VEL
LIN {X 0,Y 666.958,Z 449.856,A -85,B 0,C 180,E1 29202.506,E2 29202.506} C_VEL
LIN {X 0,Y 658.177,Z 437.007,A -85,B 0,C 180,E1 29201.452,E2 29201.452} C_VEL
LIN {X 0,Y 648.478,Z 423.923,A -85,B 0,C 180,E1 29200.245,E2 29200.245} C_VEL
LIN {X 0,Y 644.199,Z 418.398,A -85,B 0,C 180,E1 29199.696,E2 29199.696} C_VEL
LIN {X 0,Y 640.548,Z 413.525,A -85,B 0,C 180,E1 29199.213,E2 29199.213} C_VEL
LIN {X 0,Y 637.614,Z 409.778,A -85,B 0,C 180,E1 29198.82,E2 29198.82} C_VEL
LIN {X 0,Y 636.669,Z 408.252,A -85,B 0,C 180,E1 29198.687,E2 29198.687} C_VEL
LIN {X 0,Y 634.051,Z 405.66,A -85,B 0,C 180,E1 29198.342,E2 29198.342} C_VEL
LIN {X 0,Y 632.916,Z 402.597,A -85,B 0,C 180,E1 29198.155,E2 29198.155} C_VEL
LIN {X 0,Y 632.881,Z 402.368,A -85,B 0,C 180,E1 29194.995,E2 29194.995} C_VEL
LIN {X 0,Y 632.878,Z 402.392,A -85,B 0,C 180,E1 29191.787,E2 29191.787} C_VEL
LIN {X 0,Y 632.882,Z 402.388,A -85,B 0,C 180,E1 29188.705,E2 29188.705} C_VEL
LIN {X 0,Y 632.873,Z 402.363,A -85,B 0,C 180,E1 29185.551,E2 29185.551} C_VEL
LIN {X 0,Y 632.882,Z 402.392,A -85,B 0,C 180,E1 29182.443,E2 29182.443} C_VEL
LIN {X 0,Y 632.87,Z 402.376,A -85,B 0,C 180,E1 29179.281,E2 29179.281} C_VEL
LIN {X 0,Y 632.882,Z 402.379,A -85,B 0,C 180,E1 29176.239,E2 29176.239} C_VEL
LIN {X 0,Y 632.872,Z 402.384,A -85,B 0,C 180,E1 29173.151,E2 29173.151} C_VEL
LIN {X 0,Y 632.882,Z 402.37,A -85,B 0,C 180,E1 29170.008,E2 29170.008} C_VEL
LIN {X 0,Y 632.869,Z 402.387,A -85,B 0,C 180,E1 29166.896,E2 29166.896} C_VEL
LIN {X 0,Y 632.883,Z 402.366,A -85,B 0,C 180,E1 29163.805,E2 29163.805} C_VEL
LIN {X 0,Y 632.865,Z 402.389,A -85,B 0,C 180,E1 29160.634,E2 29160.634} C_VEL
LIN {X 0,Y 632.883,Z 402.363,A -85,B 0,C 180,E1 29157.555,E2 29157.555} C_VEL
LIN {X 0,Y 632.861,Z 402.391,A -85,B 0,C 180,E1 29154.378,E2 29154.378} C_VEL
LIN {X 0,Y 632.885,Z 402.362,A -85,B 0,C 180,E1 29151.368,E2 29151.368} C_VEL
LIN {X 0,Y 632.863,Z 402.393,A -85,B 0,C 180,E1 29148.24,E2 29148.24} C_VEL
LIN {X 0,Y 632.89,Z 402.363,A -85,B 0,C 180,E1 29145.171,E2 29145.171} C_VEL
LIN {X 0,Y 632.86,Z 402.396,A -85,B 0,C 180,E1 29141.961,E2 29141.961} C_VEL
LIN {X 0,Y 632.887,Z 402.37,A -85,B 0,C 180,E1 29138.887,E2 29138.887} C_VEL
LIN {X 0,Y 632.856,Z 402.382,A -85,B 0,C 180,E1 29135.745,E2 29135.745} C_VEL
LIN {X 0,Y 632.891,Z 402.398,A -85,B 0,C 180,E1 29132.629,E2 29132.629} C_VEL
LIN {X 0,Y 632.853,Z 402.375,A -85,B 0,C 180,E1 29129.524,E2 29129.524} C_VEL
LIN {X 0,Y 632.884,Z 402.368,A -85,B 0,C 180,E1 29126.533,E2 29126.533} C_VEL
LIN {X 0,Y 632.922,Z 402.617,A -85,B 0,C 180,E1 29123.957,E2 29123.957} C_VEL
LIN {X 0,Y 634.093,Z 405.749,A -85,B 0,C 180,E1 29123.524,E2 29123.524} C_VEL
LIN {X 0,Y 635.156,Z 407.3,A -85,B 0,C 180,E1 29123.256,E2 29123.256} C_VEL
LIN {X 0,Y 636.963,Z 411.054,A -85,B 0,C 180,E1 29122.704,E2 29122.704} C_VEL
LIN {X 0,Y 644.467,Z 426.425,A -85,B 0,C 180,E1 29120.555,E2 29120.555} C_VEL
LIN {X 0,Y 659.099,Z 447.415,A -85,B 0,C 180,E1 29118.706,E2 29118.706} C_VEL
LIN {X 0,Y 666.28,Z 458.234,A -85,B 0,C 180,E1 29117.844,E2 29117.844} C_VEL
LIN {X 0,Y 667.249,Z 462.966,A -85,B 0,C 180,E1 29117.679,E2 29117.679} C_VEL
LIN {X 0,Y 663.316,Z 671.494,A -85,B 0,C 180,E1 29114.847,E2 29114.847} C_VEL
LIN {X 0,Y 659.342,Z 896.455,A -85,B 0,C 180,E1 29111.871,E2 29111.871} C_VEL
LIN {X 0,Y 658.477,Z 920.939,A -85,B 0,C 180,E1 29111.474,E2 29111.474} C_VEL
LIN {X 0,Y 657.394,Z 943.793,A -85,B 0,C 180,E1 29110.981,E2 29110.981} C_VEL
LIN {X 0,Y 655.934,Z 969.606,A -85,B 0,C 180,E1 29110.275,E2 29110.275} C_VEL
LIN {X 0,Y 654.085,Z 995.654,A -85,B 0,C 180,E1 29109.378,E2 29109.378} C_VEL
LIN {X 0,Y 652.383,Z 1017.527,A -85,B 0,C 180,E1 29108.484,E2 29108.484} C_VEL
LIN {X 0,Y 650.613,Z 1038.649,A -85,B 0,C 180,E1 29107.49,E2 29107.49} C_VEL
LIN {X 0,Y 648.438,Z 1063.467,A -85,B 0,C 180,E1 29106.146,E2 29106.146} C_VEL
LIN {X 0,Y 646.233,Z 1086.282,A -85,B 0,C 180,E1 29104.71,E2 29104.71} C_VEL
LIN {X 0,Y 644.436,Z 1104.717,A -85,B 0,C 180,E1 29103.41,E2 29103.41} C_VEL
LIN {X 0,Y 642.6,Z 1123.439,A -85,B 0,C 180,E1 29101.943,E2 29101.943} C_VEL
LIN {X 0,Y 640.42,Z 1146.049,A -85,B 0,C 180,E1 29099.942,E2 29099.942} C_VEL
LIN {X 0,Y 638.837,Z 1162.888,A -85,B 0,C 180,E1 29098.262,E2 29098.262} C_VEL
LIN {X 0,Y 637.368,Z 1179.196,A -85,B 0,C 180,E1 29096.46,E2 29096.46} C_VEL
LIN {X 0,Y 635.892,Z 1197.246,A -85,B 0,C 180,E1 29094.216,E2 29094.216} C_VEL
LIN {X 0,Y 634.783,Z 1211.883,A -85,B 0,C 180,E1 29092.149,E2 29092.149} C_VEL
LIN {X 0,Y 633.916,Z 1224.709,A -85,B 0,C 180,E1 29090.115,E2 29090.115} C_VEL
LIN {X 0,Y 633.138,Z 1238.267,A -85,B 0,C 180,E1 29087.654,E2 29087.654} C_VEL
LIN {X 0,Y 632.645,Z 1248.473,A -85,B 0,C 180,E1 29085.495,E2 29085.495} C_VEL
LIN {X 0,Y 632.324,Z 1256.502,A -85,B 0,C 180,E1 29083.538,E2 29083.538} C_VEL
LIN {X 0,Y 632.155,Z 1263.345,A -85,B 0,C 180,E1 29081.592,E2 29081.592} C_VEL
LIN {X 0,Y 631.97,Z 1270.081,A -85,B 0,C 180,E1 29079.291,E2 29079.291} C_VEL
LIN {X 0,Y 631.938,Z 1275.587,A -85,B 0,C 180,E1 29076.819,E2 29076.819} C_VEL
LIN {X 0,Y 631.914,Z 1279.131,A -85,B 0,C 180,E1 29074.536,E2 29074.536} C_VEL
LIN {X 0,Y 631.907,Z 1281.147,A -85,B 0,C 180,E1 29072.362,E2 29072.362} C_VEL
LIN {X 0,Y 631.899,Z 1281.985,A -85,B 0,C 180,E1 29069.913,E2 29069.913} C_VEL
LIN {X 0,Y 631.906,Z 1281.085,A -85,B 0,C 180,E1 29067.556,E2 29067.556} C_VEL
LIN {X 0,Y 631.915,Z 1279.129,A -85,B 0,C 180,E1 29065.462,E2 29065.462} C_VEL
LIN {X 0,Y 631.939,Z 1275.602,A -85,B 0,C 180,E1 29063.189,E2 29063.189} C_VEL
LIN {X 0,Y 631.968,Z 1270.105,A -85,B 0,C 180,E1 29060.718,E2 29060.718} C_VEL
LIN {X 0,Y 632.155,Z 1263.372,A -85,B 0,C 180,E1 29058.417,E2 29058.417} C_VEL
LIN {X 0,Y 632.323,Z 1256.534,A -85,B 0,C 180,E1 29056.471,E2 29056.471} C_VEL
LIN {X 0,Y 632.644,Z 1248.511,A -85,B 0,C 180,E1 29054.513,E2 29054.513} C_VEL
LIN {X 0,Y 633.136,Z 1238.313,A -85,B 0,C 180,E1 29052.354,E2 29052.354} C_VEL
LIN {X 0,Y 633.914,Z 1224.765,A -85,B 0,C 180,E1 29049.894,E2 29049.894} C_VEL
LIN {X 0,Y 634.783,Z 1211.883,A -85,B 0,C 180,E1 29047.851,E2 29047.851} C_VEL
LIN {X 0,Y 635.898,Z 1197.185,A -85,B 0,C 180,E1 29045.776,E2 29045.776} C_VEL
LIN {X 0,Y 637.361,Z 1179.273,A -85,B 0,C 180,E1 29043.549,E2 29043.549} C_VEL
LIN {X 0,Y 638.826,Z 1163.019,A -85,B 0,C 180,E1 29041.752,E2 29041.752} C_VEL
LIN {X 0,Y 640.483,Z 1145.388,A -85,B 0,C 180,E1 29039.994,E2 29039.994} C_VEL
LIN {X 0,Y 642.591,Z 1123.548,A -85,B 0,C 180,E1 29038.066,E2 29038.066} C_VEL
LIN {X 0,Y 644.433,Z 1104.719,A -85,B 0,C 180,E1 29036.59,E2 29036.59} C_VEL
LIN {X 0,Y 646.219,Z 1086.409,A -85,B 0,C 180,E1 29035.299,E2 29035.299} C_VEL
LIN {X 0,Y 648.42,Z 1063.613,A -85,B 0,C 180,E1 29033.863,E2 29033.863} C_VEL
LIN {X 0,Y 650.599,Z 1038.837,A -85,B 0,C 180,E1 29032.519,E2 29032.519} C_VEL
LIN {X 0,Y 652.365,Z 1017.737,A -85,B 0,C 180,E1 29031.525,E2 29031.525} C_VEL
LIN {X 0,Y 654.064,Z 995.889,A -85,B 0,C 180,E1 29030.631,E2 29030.631} C_VEL
LIN {X 0,Y 655.993,Z 968.642,A -85,B 0,C 180,E1 29029.695,E2 29029.695} C_VEL
LIN {X 0,Y 657.406,Z 943.527,A -85,B 0,C 180,E1 29029.012,E2 29029.012} C_VEL
LIN {X 0,Y 658.492,Z 920.605,A -85,B 0,C 180,E1 29028.52,E2 29028.52} C_VEL
LIN {X 0,Y 659.386,Z 895.085,A -85,B 0,C 180,E1 29028.109,E2 29028.109} C_VEL
LIN {X 0,Y 663.357,Z 669.221,A -85,B 0,C 180,E1 29025.123,E2 29025.123} C_VEL
LIN {X 0,Y 667.262,Z 462.247,A -85,B 0,C 180,E1 29022.311,E2 29022.311} C_VEL
LIN {X 0,Y 665.873,Z 457.34,A -85,B 0,C 180,E1 29022.104,E2 29022.104} C_VEL
LIN {X 0,Y 651.703,Z 436.87,A -85,B 0,C 180,E1 29020.38,E2 29020.38} C_VEL
LIN {X 0,Y 644.123,Z 425.799,A -85,B 0,C 180,E1 29019.381,E2 29019.381} C_VEL
LIN {X 0,Y 636.948,Z 411.074,A -85,B 0,C 180,E1 29017.297,E2 29017.297} C_VEL
LIN {X 0,Y 635.088,Z 407.096,A -85,B 0,C 180,E1 29016.719,E2 29016.719} C_VEL
LIN {X 0,Y 633.214,Z 403.868,A -85,B 0,C 180,E1 29016.198,E2 29016.198} C_VEL
LIN {X 0,Y 632.896,Z 402.393,A -85,B 0,C 180,E1 29015.995,E2 29015.995} C_VEL
LIN {X 0,Y 632.822,Z 402.384,A -85,B 0,C 180,E1 29012.978,E2 29012.978} C_VEL
LIN {X 0,Y 632.881,Z 402.367,A -85,B 0,C 180,E1 29010.042,E2 29010.042} C_VEL
LIN {X 0,Y 632.823,Z 402.398,A -85,B 0,C 180,E1 29006.967,E2 29006.967} C_VEL
LIN {X 0,Y 632.836,Z 402.383,A -85,B 0,C 180,E1 29004.156,E2 29004.156} C_VEL
LIN {X 0,Y 632.82,Z 402.376,A -85,B 0,C 180,E1 29000.983,E2 29000.983} C_VEL
LIN {X 0,Y 632.808,Z 402.399,A -85,B 0,C 180,E1 28998.286,E2 28998.286} C_VEL
LIN {X 0,Y 632.849,Z 402.367,A -85,B 0,C 180,E1 28995.205,E2 28995.205} C_VEL
LIN {X 0,Y 632.792,Z 402.404,A -85,B 0,C 180,E1 28992.41,E2 28992.41} C_VEL
LIN {X 0,Y 632.841,Z 402.37,A -85,B 0,C 180,E1 28989.55,E2 28989.55} C_VEL
LIN {X 0,Y 632.793,Z 402.405,A -85,B 0,C 180,E1 28986.533,E2 28986.533} C_VEL
LIN {X 0,Y 632.793,Z 402.38,A -85,B 0,C 180,E1 28983.896,E2 28983.896} C_VEL
LIN {X 0,Y 632.85,Z 402.399,A -85,B 0,C 180,E1 28980.815,E2 28980.815} C_VEL
LIN {X 0,Y 632.797,Z 402.384,A -85,B 0,C 180,E1 28978.008,E2 28978.008} C_VEL
LIN {X 0,Y 632.868,Z 402.386,A -85,B 0,C 180,E1 28975.106,E2 28975.106} C_VEL
LIN {X 0,Y 632.812,Z 402.385,A -85,B 0,C 180,E1 28972.099,E2 28972.099} C_VEL
LIN {X 0,Y 632.83,Z 402.387,A -85,B 0,C 180,E1 28969.347,E2 28969.347} C_VEL
LIN {X 0,Y 632.832,Z 402.38,A -85,B 0,C 180,E1 28966.104,E2 28966.104} C_VEL
LIN {X 0,Y 632.827,Z 402.391,A -85,B 0,C 180,E1 28963.382,E2 28963.382} C_VEL
LIN {X 0,Y 632.873,Z 402.367,A -85,B 0,C 180,E1 28960.239,E2 28960.239} C_VEL
LIN {X 0,Y 632.835,Z 402.398,A -85,B 0,C 180,E1 28957.31,E2 28957.31} C_VEL
LIN {X 0,Y 632.887,Z 402.365,A -85,B 0,C 180,E1 28954.212,E2 28954.212} C_VEL
LIN {X 0,Y 632.841,Z 402.397,A -85,B 0,C 180,E1 28951.19,E2 28951.19} C_VEL
LIN {X 0,Y 632.892,Z 402.386,A -85,B 0,C 180,E1 28948.151,E2 28948.151} C_VEL
LIN {X 0,Y 632.845,Z 402.37,A -85,B 0,C 180,E1 28945.074,E2 28945.074} C_VEL
LIN {X 0,Y 632.888,Z 402.368,A -85,B 0,C 180,E1 28942.022,E2 28942.022} C_VEL
LIN {X 0,Y 632.912,Z 402.548,A -85,B 0,C 180,E1 28941.755,E2 28941.755} C_VEL
LIN {X 0,Y 634.099,Z 405.73,A -85,B 0,C 180,E1 28941.561,E2 28941.561} C_VEL
LIN {X 0,Y 636.798,Z 408.315,A -85,B 0,C 180,E1 28941.207,E2 28941.207} C_VEL
LIN {X 0,Y 639.666,Z 412.676,A -85,B 0,C 180,E1 28940.809,E2 28940.809} C_VEL
LIN {X 0,Y 641.59,Z 414.796,A -85,B 0,C 180,E1 28940.56,E2 28940.56} C_VEL
LIN {X 0,Y 644.911,Z 419.104,A -85,B 0,C 180,E1 28940.126,E2 28940.126} C_VEL
LIN {X 0,Y 657.651,Z 436.276,A -85,B 0,C 180,E1 28938.522,E2 28938.522} C_VEL
LIN {X 0,Y 665.137,Z 447.085,A -85,B 0,C 180,E1 28937.62,E2 28937.62} C_VEL
LIN {X 0,Y 666.952,Z 450.118,A -85,B 0,C 180,E1 28937.401,E2 28937.401} C_VEL
LIN {X 0,Y 666.637,Z 466.438,A -85,B 0,C 180,E1 28937.175,E2 28937.175} C_VEL
LIN {X 0,Y 665.806,Z 474.143,A -85,B 0,C 180,E1 28937.133,E2 28937.133} C_VEL
LIN {X 0,Y 661.135,Z 494.828,A -85,B 0,C 180,E1 28937.248,E2 28937.248} C_VEL
LIN {X 0,Y 660.474,Z 501.439,A -85,B 0,C 180,E1 28937.206,E2 28937.206} C_VEL
LIN {X 0,Y 656.211,Z 716.186,A -85,B 0,C 180,E1 28934.292,E2 28934.292} C_VEL
LIN {X 0,Y 653.109,Z 874.818,A -85,B 0,C 180,E1 28932.173,E2 28932.173} C_VEL
LIN {X 0,Y 652.007,Z 901.858,A -85,B 0,C 180,E1 28931.682,E2 28931.682} C_VEL
LIN {X 0,Y 650.459,Z 928.226,A -85,B 0,C 180,E1 28931.024,E2 28931.024} C_VEL
LIN {X 0,Y 648.966,Z 950.148,A -85,B 0,C 180,E1 28930.345,E2 28930.345} C_VEL
LIN {X 0,Y 647.457,Z 970.018,A -85,B 0,C 180,E1 28929.621,E2 28929.621} C_VEL
LIN {X 0,Y 645.614,Z 992.116,A -85,B 0,C 180,E1 28928.687,E2 28928.687} C_VEL
LIN {X 0,Y 643.197,Z 1018.627,A -85,B 0,C 180,E1 28927.369,E2 28927.369} C_VEL
LIN {X 0,Y 641.122,Z 1039.439,A -85,B 0,C 180,E1 28926.171,E2 28926.171} C_VEL
LIN {X 0,Y 639.179,Z 1058.43,A -85,B 0,C 180,E1 28924.944,E2 28924.944} C_VEL
LIN {X 0,Y 637.176,Z 1077.593,A -85,B 0,C 180,E1 28923.563,E2 28923.563} C_VEL
LIN {X 0,Y 634.791,Z 1100.207,A -85,B 0,C 180,E1 28921.725,E2 28921.725} C_VEL
LIN {X 0,Y 632.891,Z 1118.591,A -85,B 0,C 180,E1 28920.028,E2 28920.028} C_VEL
LIN {X 0,Y 631.252,Z 1134.881,A -85,B 0,C 180,E1 28918.365,E2 28918.365} C_VEL
LIN {X 0,Y 629.501,Z 1153.101,A -85,B 0,C 180,E1 28916.299,E2 28916.299} C_VEL
LIN {X 0,Y 628.032,Z 1169.71,A -85,B 0,C 180,E1 28914.147,E2 28914.147} C_VEL
LIN {X 0,Y 626.958,Z 1183.125,A -85,B 0,C 180,E1 28912.202,E2 28912.202} C_VEL
LIN {X 0,Y 625.954,Z 1197.361,A -85,B 0,C 180,E1 28909.886,E2 28909.886} C_VEL
LIN {X 0,Y 625.167,Z 1209.958,A -85,B 0,C 180,E1 28907.493,E2 28907.493} C_VEL
LIN {X 0,Y 624.676,Z 1219.543,A -85,B 0,C 180,E1 28905.404,E2 28905.404} C_VEL
LIN {X 0,Y 624.34,Z 1227.777,A -85,B 0,C 180,E1 28903.328,E2 28903.328} C_VEL
LIN {X 0,Y 624.099,Z 1236.152,A -85,B 0,C 180,E1 28900.799,E2 28900.799} C_VEL
LIN {X 0,Y 623.991,Z 1242.437,A -85,B 0,C 180,E1 28898.38,E2 28898.38} C_VEL
LIN {X 0,Y 623.936,Z 1246.966,A -85,B 0,C 180,E1 28896.067,E2 28896.067} C_VEL
LIN {X 0,Y 623.913,Z 1250.237,A -85,B 0,C 180,E1 28893.579,E2 28893.579} C_VEL
LIN {X 0,Y 623.893,Z 1251.704,A -85,B 0,C 180,E1 28891.19,E2 28891.19} C_VEL
LIN {X 0,Y 623.864,Z 1251.837,A -85,B 0,C 180,E1 28889.261,E2 28889.261} C_VEL
LIN {X 0,Y 623.906,Z 1250.977,A -85,B 0,C 180,E1 28887.332,E2 28887.332} C_VEL
LIN {X 0,Y 623.913,Z 1248.95,A -85,B 0,C 180,E1 28885.216,E2 28885.216} C_VEL
LIN {X 0,Y 623.952,Z 1245.155,A -85,B 0,C 180,E1 28882.816,E2 28882.816} C_VEL
LIN {X 0,Y 623.989,Z 1239.695,A -85,B 0,C 180,E1 28880.403,E2 28880.403} C_VEL
